KUKA KRL program: MyProgram_016().src

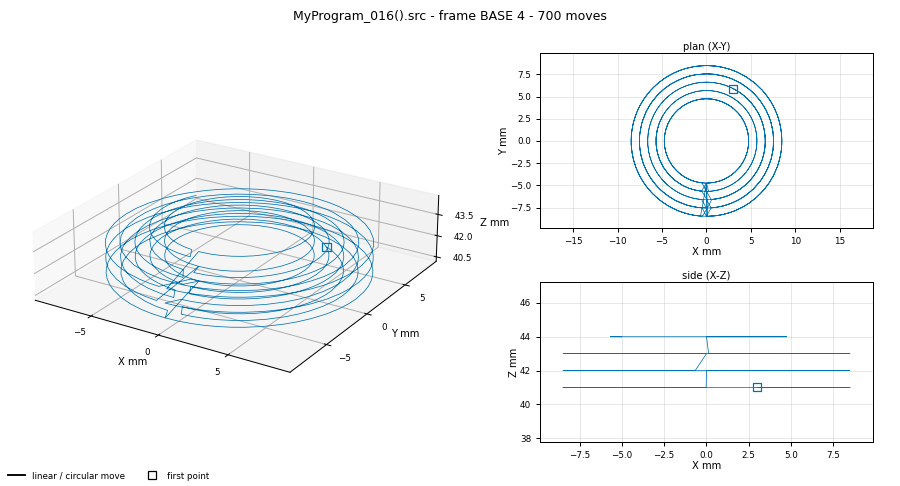
[picture p0: tool path of MyProgram_016().src in frame BASE 4, 700 of 700 moves have a stored position in this frame; points joined in program order, loops and branches not executed]
&ACCESS RVP
&REL 1
&PARAM TEMPLATE = C:\KRC\Roboter\Template\vorgabe
&PARAM EDITMASK = *
DEF MyProgram_016()
; ---- Setting reference (Base) ----
$BASE = BASE_DATA[4]

; --------------------------
; ---- Setting tool (TCP) ----
$TOOL = TOOL_DATA[3]
; --------------------------

$VEL.CP = VEL_APROX_PRINT
Startdeposition()
$VEL.CP = VEL_PRINT
LIN {X 3.0027,Y 5.8982,Z 41,A -2.319,B 0,C 0,E1 0.1598,E2 90.0724} C_DIS
LIN {X 3.6295,Y 5.5354,Z 41,A -2.3113,B 0,C 0,E1 0.1598,E2 90.0724} C_DIS
LIN {X 4.2131,Y 5.1066,Z 41,A -2.308,B 0,C 0,E1 0.1598,E2 90.0724} C_DIS
LIN {X 4.7456,Y 4.6156,Z 41,A -2.3092,B 0,C 0,E1 0.1598,E2 90.0724} C_DIS
LIN {X 5.2207,Y 4.0691,Z 41,A -2.3149,B 0,C 0,E1 0.1598,E2 90.0723} C_DIS
LIN {X 5.6347,Y 3.4746,Z 41,A -2.3249,B 0,C 0,E1 0.1598,E2 90.0723} C_DIS
LIN {X 5.9818,Y 2.8391,Z 41,A -2.3392,B 0,C 0,E1 0.1598,E2 90.0723} C_DIS
LIN {X 6.2545,Y 2.1682,Z 41,A -2.3577,B 0,C 0,E1 0.1598,E2 90.0722} C_DIS
LIN {X 6.4955,Y 1.2955,Z 41,A -2.3857,B 0,C 0,E1 0.1598,E2 90.0719} C_DIS
LIN {X 6.6144,Y 0.2312,Z 41,A -2.4266,B 0,C 0,E1 0.1598,E2 90.0717} C_DIS
LIN {X 6.5984,Y -0.514,Z 41,A -2.4593,B 0,C 0,E1 0.1598,E2 90.072} C_DIS
LIN {X 6.4986,Y -1.2526,Z 41,A -2.4944,B 0,C 0,E1 0.1598,E2 90.072} C_DIS
LIN {X 6.3195,Y -1.9763,Z 41,A -2.5319,B 0,C 0,E1 0.1598,E2 90.072} C_DIS
LIN {X 6.0549,Y -2.6732,Z 41,A -2.5714,B 0,C 0,E1 0.1598,E2 90.0719} C_DIS
LIN {X 5.7165,Y -3.3374,Z 41,A -2.6122,B 0,C 0,E1 0.1598,E2 90.0719} C_DIS
LIN {X 5.3054,Y -3.9593,Z 41,A -2.6538,B 0,C 0,E1 0.1598,E2 90.0719} C_DIS
LIN {X 4.8275,Y -4.5316,Z 41,A -2.6958,B 0,C 0,E1 0.1598,E2 90.0719} C_DIS
LIN {X 4.2857,Y -5.0436,Z 41,A -2.7375,B 0,C 0,E1 0.1598,E2 90.0718} C_DIS
LIN {X 3.691,Y -5.4931,Z 41,A -2.7785,B 0,C 0,E1 0.1598,E2 90.0718} C_DIS
LIN {X 3.0503,Y -5.874,Z 41,A -2.8183,B 0,C 0,E1 0.1598,E2 90.0718} C_DIS
LIN {X 2.3699,Y -6.1782,Z 41,A -2.8563,B 0,C 0,E1 0.1598,E2 90.0718} C_DIS
LIN {X 1.6605,Y -6.4069,Z 41,A -2.892,B 0,C 0,E1 0.1598,E2 90.0717} C_DIS
LIN {X 0.9297,Y -6.5533,Z 41,A -2.9251,B 0,C 0,E1 0.1598,E2 90.0717} C_DIS
LIN {X 0.0006,Y -6.6224,Z 41,A -2.9621,B 0,C 0,E1 0.1598,E2 90.0717} C_DIS
Enddeposition()
LIN {X 0.0006,Y -6.6224,Z 41,A -2.9621,B 0,C 0,E1 0.1598,E2 90.0717} C_DIS
Startdeposition()
$VEL.CP = VEL_PRINT
LIN {X 0.5218,Y -7.5346,Z 41,A -2.9814,B 0,C 0,E1 0.1598,E2 90.071} C_DIS
LIN {X 1.2142,Y -7.4561,Z 41,A -2.9532,B 0,C 0,E1 0.1598,E2 90.0716} C_DIS
LIN {X 1.8961,Y -7.3127,Z 41,A -2.9222,B 0,C 0,E1 0.1598,E2 90.0716} C_DIS
LIN {X 2.7263,Y -7.0488,Z 41,A -2.8805,B 0,C 0,E1 0.1598,E2 90.0716} C_DIS
LIN {X 3.6839,Y -6.5978,Z 41,A -2.8261,B 0,C 0,E1 0.1598,E2 90.0717} C_DIS
LIN {X 4.3969,Y -6.1467,Z 41,A -2.7807,B 0,C 0,E1 0.1598,E2 90.0717} C_DIS
LIN {X 5.2728,Y -5.4135,Z 41,A -2.7171,B 0,C 0,E1 0.1598,E2 90.0717} C_DIS
LIN {X 6.0845,Y -4.4837,Z 41,A -2.6475,B 0,C 0,E1 0.1598,E2 90.0717} C_DIS
LIN {X 6.5832,Y -3.7041,Z 41,A -2.596,B 0,C 0,E1 0.1598,E2 90.0718} C_DIS
LIN {X 6.9129,Y -3.0412,Z 41,A -2.5557,B 0,C 0,E1 0.1598,E2 90.0719} C_DIS
LIN {X 7.287,Y -2.0035,Z 41,A -2.4973,B 0,C 0,E1 0.1598,E2 90.0717} C_DIS
LIN {X 7.4913,Y -1.0048,Z 41,A -2.4471,B 0,C 0,E1 0.1598,E2 90.0717} C_DIS
LIN {X 7.5586,Y -0.0079,Z 41,A -2.4022,B 0,C 0,E1 0.1598,E2 90.0718} C_DIS
LIN {X 7.499,Y 0.937,Z 41,A -2.3641,B 0,C 0,E1 0.1598,E2 90.0719} C_DIS
LIN {X 7.2647,Y 2.068,Z 41,A -2.3242,B 0,C 0,E1 0.1598,E2 90.0717} C_DIS
LIN {X 7.0052,Y 2.8257,Z 41,A -2.3019,B 0,C 0,E1 0.1598,E2 90.0721} C_DIS
LIN {X 6.6657,Y 3.5511,Z 41,A -2.2835,B 0,C 0,E1 0.1598,E2 90.0722} C_DIS
LIN {X 6.0442,Y 4.5361,Z 41,A -2.2642,B 0,C 0,E1 0.1598,E2 90.072} C_DIS
LIN {X 5.3435,Y 5.346,Z 41,A -2.2557,B 0,C 0,E1 0.1598,E2 90.0722} C_DIS
LIN {X 4.6544,Y 5.9486,Z 41,A -2.2557,B 0,C 0,E1 0.1598,E2 90.0723} C_DIS
LIN {X 3.7373,Y 6.5685,Z 41,A -2.2631,B 0,C 0,E1 0.1598,E2 90.0723} C_DIS
LIN {X 2.7804,Y 7.0216,Z 41,A -2.2793,B 0,C 0,E1 0.1598,E2 90.0723} C_DIS
LIN {X 1.9771,Y 7.2898,Z 41,A -2.2976,B 0,C 0,E1 0.1598,E2 90.0725} C_DIS
LIN {X 0.8628,Y 7.5074,Z 41,A -2.3295,B 0,C 0,E1 0.1598,E2 90.0725} C_DIS
LIN {X -0.0807,Y 7.557,Z 41,A -2.3623,B 0,C 0,E1 0.1598,E2 90.0725} C_DIS
LIN {X -1.2554,Y 7.4477,Z 41,A -2.4103,B 0,C 0,E1 0.1598,E2 90.0724} C_DIS
LIN {X -2.007,Y 7.2809,Z 41,A -2.4451,B 0,C 0,E1 0.1598,E2 90.0723} C_DIS
LIN {X -2.7375,Y 7.0382,Z 41,A -2.4823,B 0,C 0,E1 0.1598,E2 90.0723} C_DIS
LIN {X -3.9575,Y 6.4373,Z 41,A -2.5526,B 0,C 0,E1 0.1598,E2 90.072} C_DIS
LIN {X -4.6822,Y 5.9317,Z 41,A -2.6008,B 0,C 0,E1 0.1598,E2 90.072} C_DIS
LIN {X -5.4823,Y 5.2003,Z 41,A -2.6611,B 0,C 0,E1 0.1598,E2 90.0718} C_DIS
LIN {X -6.1884,Y 4.3366,Z 41,A -2.7235,B 0,C 0,E1 0.1598,E2 90.0716} C_DIS
LIN {X -6.7771,Y 3.3427,Z 41,A -2.7871,B 0,C 0,E1 0.1598,E2 90.0714} C_DIS
LIN {X -7.2905,Y 1.9898,Z 41,A -2.8628,B 0,C 0,E1 0.1598,E2 90.0708} C_DIS
LIN {X -7.5205,Y 0.6986,Z 41,A -2.9259,B 0,C 0,E1 0.1598,E2 90.0708} C_DIS
LIN {X -7.5526,Y -0.1182,Z 41,A -2.9621,B 0,C 0,E1 0.1598,E2 90.0712} C_DIS
LIN {X -7.4933,Y -0.9334,Z 41,A -2.9944,B 0,C 0,E1 0.1598,E2 90.0712} C_DIS
LIN {X -7.3508,Y -1.7381,Z 41,A -3.0233,B 0,C 0,E1 0.1598,E2 90.0712} C_DIS
LIN {X -7.0039,Y -2.8395,Z 41,A -3.0569,B 0,C 0,E1 0.1598,E2 90.0709} C_DIS
LIN {X -6.6343,Y -3.6177,Z 41,A -3.0765,B 0,C 0,E1 0.1598,E2 90.0712} C_DIS
LIN {X -5.9525,Y -4.6552,Z 41,A -3.0952,B 0,C 0,E1 0.1598,E2 90.0708} C_DIS
LIN {X -5.2119,Y -5.4671,Z 41,A -3.1027,B 0,C 0,E1 0.1598,E2 90.0711} C_DIS
LIN {X -4.6479,Y -5.9517,Z 41,A -3.1027,B 0,C 0,E1 0.1598,E2 90.0713} C_DIS
LIN {X -4.0412,Y -6.3817,Z 41,A -3.0988,B 0,C 0,E1 0.1598,E2 90.0713} C_DIS
LIN {X -3.394,Y -6.7479,Z 41,A -3.0906,B 0,C 0,E1 0.1598,E2 90.0713} C_DIS
LIN {X -2.388,Y -7.1707,Z 41,A -3.0717,B 0,C 0,E1 0.1598,E2 90.0713} C_DIS
LIN {X -1.4895,Y -7.4088,Z 41,A -3.0489,B 0,C 0,E1 0.1598,E2 90.0715} C_DIS
LIN {X -0.4781,Y -7.5384,Z 41,A -3.0174,B 0,C 0,E1 0.1598,E2 90.0715} C_DIS
LIN {X -0.4781,Y -7.5384,Z 41,A -3.0174,B 0,C 0,E1 0.1598,E2 90.0715} C_DIS
Enddeposition()
LIN {X -0.0182,Y -8.489,Z 41,A -3.04,B 0,C 0,E1 0.1598,E2 90.0703} C_DIS
Startdeposition()
$VEL.CP = VEL_PRINT
LIN {X -1.0751,Y -8.4193,Z 41,A -3.0769,B 0,C 0,E1 0.1598,E2 90.0714} C_DIS
LIN {X -1.9094,Y -8.27,Z 41,A -3.1012,B 0,C 0,E1 0.1598,E2 90.0714} C_DIS
LIN {X -2.9255,Y -7.9703,Z 41,A -3.1256,B 0,C 0,E1 0.1598,E2 90.0714} C_DIS
LIN {X -3.9562,Y -7.5135,Z 41,A -3.1439,B 0,C 0,E1 0.1598,E2 90.0712} C_DIS
LIN {X -5.0038,Y -6.8555,Z 41,A -3.1543,B 0,C 0,E1 0.1598,E2 90.0712} C_DIS
LIN {X -5.667,Y -6.3182,Z 41,A -3.1559,B 0,C 0,E1 0.1598,E2 90.0712} C_DIS
LIN {X -6.273,Y -5.7172,Z 41,A -3.1526,B 0,C 0,E1 0.1598,E2 90.0712} C_DIS
LIN {X -6.8156,Y -5.0583,Z 41,A -3.1445,B 0,C 0,E1 0.1598,E2 90.0712} C_DIS
LIN {X -7.2893,Y -4.3483,Z 41,A -3.1318,B 0,C 0,E1 0.1598,E2 90.0712} C_DIS
LIN {X -7.6893,Y -3.5943,Z 41,A -3.1145,B 0,C 0,E1 0.1598,E2 90.0712} C_DIS
LIN {X -8.0114,Y -2.8039,Z 41,A -3.0929,B 0,C 0,E1 0.1598,E2 90.0712} C_DIS
LIN {X -8.2523,Y -1.9851,Z 41,A -3.0671,B 0,C 0,E1 0.1598,E2 90.0712} C_DIS
LIN {X -8.4389,Y -0.9347,Z 41,A -3.0292,B 0,C 0,E1 0.1598,E2 90.0709} C_DIS
LIN {X -8.4896,Y 0.137,Z 41,A -2.9857,B 0,C 0,E1 0.1598,E2 90.0709} C_DIS
LIN {X -8.4116,Y 1.1667,Z 41,A -2.9394,B 0,C 0,E1 0.1598,E2 90.0711} C_DIS
LIN {X -8.1845,Y 2.2482,Z 41,A -2.8853,B 0,C 0,E1 0.1598,E2 90.0711} C_DIS
LIN {X -7.7971,Y 3.36,Z 41,A -2.824,B 0,C 0,E1 0.1598,E2 90.0712} C_DIS
LIN {X -7.21,Y 4.483,Z 41,A -2.7549,B 0,C 0,E1 0.1598,E2 90.0712} C_DIS
LIN {X -6.5678,Y 5.3748,Z 41,A -2.6937,B 0,C 0,E1 0.1598,E2 90.0716} C_DIS
LIN {X -5.9685,Y 6.0403,Z 41,A -2.6436,B 0,C 0,E1 0.1598,E2 90.0718} C_DIS
LIN {X -5.0746,Y 6.8036,Z 41,A -2.5784,B 0,C 0,E1 0.1598,E2 90.0718} C_DIS
LIN {X -4.3639,Y 7.2802,Z 41,A -2.5321,B 0,C 0,E1 0.1598,E2 90.0721} C_DIS
LIN {X -3.6087,Y 7.6827,Z 41,A -2.4873,B 0,C 0,E1 0.1598,E2 90.0721} C_DIS
LIN {X -2.8167,Y 8.0069,Z 41,A -2.4444,B 0,C 0,E1 0.1598,E2 90.0723} C_DIS
LIN {X -1.9961,Y 8.2497,Z 41,A -2.4038,B 0,C 0,E1 0.1598,E2 90.0723} C_DIS
LIN {X -1.1553,Y 8.4087,Z 41,A -2.366,B 0,C 0,E1 0.1598,E2 90.0724} C_DIS
LIN {X -0.0888,Y 8.4907,Z 41,A -2.3232,B 0,C 0,E1 0.1598,E2 90.0724} C_DIS
LIN {X 1.0545,Y 8.4223,Z 41,A -2.2839,B 0,C 0,E1 0.1598,E2 90.0725} C_DIS
LIN {X 1.8987,Y 8.2723,Z 41,A -2.2591,B 0,C 0,E1 0.1598,E2 90.0725} C_DIS
LIN {X 2.7237,Y 8.0385,Z 41,A -2.2385,B 0,C 0,E1 0.1598,E2 90.0725} C_DIS
LIN {X 3.5208,Y 7.7226,Z 41,A -2.2225,B 0,C 0,E1 0.1598,E2 90.0725} C_DIS
LIN {X 4.4673,Y 7.2197,Z 41,A -2.2088,B 0,C 0,E1 0.1598,E2 90.0725} C_DIS
LIN {X 5.5023,Y 6.4657,Z 41,A -2.2025,B 0,C 0,E1 0.1598,E2 90.0723} C_DIS
LIN {X 6.2699,Y 5.7205,Z 41,A -2.2059,B 0,C 0,E1 0.1598,E2 90.0723} C_DIS
LIN {X 6.8143,Y 5.0601,Z 41,A -2.214,B 0,C 0,E1 0.1598,E2 90.0723} C_DIS
LIN {X 7.2893,Y 4.3481,Z 41,A -2.2268,B 0,C 0,E1 0.1598,E2 90.0723} C_DIS
LIN {X 7.6903,Y 3.592,Z 41,A -2.2442,B 0,C 0,E1 0.1598,E2 90.0723} C_DIS
LIN {X 8.0125,Y 2.7991,Z 41,A -2.2661,B 0,C 0,E1 0.1598,E2 90.0722} C_DIS
LIN {X 8.2538,Y 1.978,Z 41,A -2.2922,B 0,C 0,E1 0.1598,E2 90.0722} C_DIS
LIN {X 8.4112,Y 1.1367,Z 41,A -2.3223,B 0,C 0,E1 0.1598,E2 90.0721} C_DIS
LIN {X 8.4922,Y -0.0058,Z 41,A -2.3678,B 0,C 0,E1 0.1598,E2 90.0717} C_DIS
LIN {X 8.4473,Y -0.8607,Z 41,A -2.406,B 0,C 0,E1 0.1598,E2 90.0717} C_DIS
LIN {X 8.3172,Y -1.7063,Z 41,A -2.4471,B 0,C 0,E1 0.1598,E2 90.0719} C_DIS
LIN {X 8.0233,Y -2.7811,Z 41,A -2.5036,B 0,C 0,E1 0.1598,E2 90.0717} C_DIS
LIN {X 7.5387,Y -3.8974,Z 41,A -2.5689,B 0,C 0,E1 0.1598,E2 90.0714} C_DIS
LIN {X 7.0759,Y -4.6845,Z 41,A -2.6199,B 0,C 0,E1 0.1598,E2 90.0717} C_DIS
LIN {X 6.5318,Y -5.4179,Z 41,A -2.6712,B 0,C 0,E1 0.1598,E2 90.0717} C_DIS
LIN {X 5.6483,Y -6.3408,Z 41,A -2.7429,B 0,C 0,E1 0.1598,E2 90.0715} C_DIS
LIN {X 4.7399,Y -7.0403,Z 41,A -2.8062,B 0,C 0,E1 0.1598,E2 90.0715} C_DIS
LIN {X 4.0492,Y -7.4582,Z 41,A -2.8495,B 0,C 0,E1 0.1598,E2 90.0717} C_DIS
LIN {X 3.3221,Y -7.8087,Z 41,A -2.8911,B 0,C 0,E1 0.1598,E2 90.0717} C_DIS
LIN {X 2.5651,Y -8.0886,Z 41,A -2.9308,B 0,C 0,E1 0.1598,E2 90.0717} C_DIS
LIN {X 1.785,Y -8.2955,Z 41,A -2.9683,B 0,C 0,E1 0.1598,E2 90.0717} C_DIS
LIN {X 0.9888,Y -8.4278,Z 41,A -3.0031,B 0,C 0,E1 0.1598,E2 90.0716} C_DIS
LIN {X -0.0182,Y -8.489,Z 41,A -3.0426,B 0,C 0,E1 0.1598,E2 90.0716} C_DIS
Enddeposition()
LIN {X 0.0009,Y -4.7546,Z 42,A -2.8683,B 0,C 0,E1 0.1598,E2 90.0604} C_DIS
Startdeposition()
$VEL.CP = VEL_PRINT
LIN {X 0.0009,Y -4.7546,Z 42,A -2.8741,B 0,C 0,E1 0.1598,E2 90.0661} C_DIS
LIN {X 0.8353,Y -4.6792,Z 42,A -2.8451,B 0,C 0,E1 0.1598,E2 90.0711} C_DIS
LIN {X 1.4852,Y -4.5142,Z 42,A -2.8149,B 0,C 0,E1 0.1598,E2 90.0718} C_DIS
LIN {X 2.1053,Y -4.2593,Z 42,A -2.7813,B 0,C 0,E1 0.1598,E2 90.0718} C_DIS
LIN {X 2.7516,Y -3.8714,Z 42,A -2.741,B 0,C 0,E1 0.1598,E2 90.0718} C_DIS
LIN {X 3.2075,Y -3.5024,Z 42,A -2.7085,B 0,C 0,E1 0.1598,E2 90.0719} C_DIS
LIN {X 3.671,Y -3.0181,Z 42,A -2.6708,B 0,C 0,E1 0.1598,E2 90.0719} C_DIS
LIN {X 4.0596,Y -2.4718,Z 42,A -2.6332,B 0,C 0,E1 0.1598,E2 90.0719} C_DIS
LIN {X 4.3647,Y -1.8749,Z 42,A -2.5966,B 0,C 0,E1 0.1598,E2 90.0719} C_DIS
LIN {X 4.5854,Y -1.2421,Z 42,A -2.5614,B 0,C 0,E1 0.1598,E2 90.0719} C_DIS
LIN {X 4.7151,Y -0.5846,Z 42,A -2.5286,B 0,C 0,E1 0.1598,E2 90.0719} C_DIS
LIN {X 4.7506,Y 0.0847,Z 42,A -2.4988,B 0,C 0,E1 0.1598,E2 90.0719} C_DIS
LIN {X 4.6913,Y 0.7523,Z 42,A -2.4725,B 0,C 0,E1 0.1598,E2 90.072} C_DIS
LIN {X 4.539,Y 1.405,Z 42,A -2.4504,B 0,C 0,E1 0.1598,E2 90.072} C_DIS
LIN {X 4.2971,Y 2.0303,Z 42,A -2.4327,B 0,C 0,E1 0.1598,E2 90.072} C_DIS
LIN {X 3.9682,Y 2.6145,Z 42,A -2.4199,B 0,C 0,E1 0.1598,E2 90.0721} C_DIS
LIN {X 3.5592,Y 3.1456,Z 42,A -2.4124,B 0,C 0,E1 0.1598,E2 90.0721} C_DIS
LIN {X 3.0809,Y 3.6151,Z 42,A -2.4101,B 0,C 0,E1 0.1598,E2 90.0722} C_DIS
LIN {X 2.5429,Y 4.0149,Z 42,A -2.413,B 0,C 0,E1 0.1598,E2 90.0722} C_DIS
LIN {X 1.8748,Y 4.3642,Z 42,A -2.4228,B 0,C 0,E1 0.1598,E2 90.0722} C_DIS
LIN {X 1.3227,Y 4.562,Z 42,A -2.4348,B 0,C 0,E1 0.1598,E2 90.0722} C_DIS
LIN {X 0.6678,Y 4.7047,Z 42,A -2.4529,B 0,C 0,E1 0.1598,E2 90.0722} C_DIS
LIN {X -0.0009,Y 4.7506,Z 42,A -2.4756,B 0,C 0,E1 0.1598,E2 90.0722} C_DIS
LIN {X -0.6694,Y 4.7033,Z 42,A -2.5022,B 0,C 0,E1 0.1598,E2 90.0722} C_DIS
LIN {X -1.3245,Y 4.5621,Z 42,A -2.5324,B 0,C 0,E1 0.1598,E2 90.0722} C_DIS
LIN {X -1.9536,Y 4.331,Z 42,A -2.5653,B 0,C 0,E1 0.1598,E2 90.0722} C_DIS
LIN {X -2.5432,Y 4.0123,Z 42,A -2.6005,B 0,C 0,E1 0.1598,E2 90.0721} C_DIS
LIN {X -3.0824,Y 3.6143,Z 42,A -2.6372,B 0,C 0,E1 0.1598,E2 90.072} C_DIS
LIN {X -3.561,Y 3.145,Z 42,A -2.6747,B 0,C 0,E1 0.1598,E2 90.0719} C_DIS
LIN {X -3.9685,Y 2.6128,Z 42,A -2.7122,B 0,C 0,E1 0.1598,E2 90.0719} C_DIS
LIN {X -4.2978,Y 2.0289,Z 42,A -2.7491,B 0,C 0,E1 0.1598,E2 90.0717} C_DIS
LIN {X -4.5408,Y 1.404,Z 42,A -2.7845,B 0,C 0,E1 0.1598,E2 90.0717} C_DIS
LIN {X -4.6932,Y 0.7511,Z 42,A -2.8177,B 0,C 0,E1 0.1598,E2 90.0716} C_DIS
LIN {X -4.7509,Y 0.0831,Z 42,A -2.8481,B 0,C 0,E1 0.1598,E2 90.0716} C_DIS
LIN {X -4.7165,Y -0.5864,Z 42,A -2.8752,B 0,C 0,E1 0.1598,E2 90.0716} C_DIS
LIN {X -4.5857,Y -1.2439,Z 42,A -2.8983,B 0,C 0,E1 0.1598,E2 90.0715} C_DIS
LIN {X -4.3651,Y -1.8769,Z 42,A -2.917,B 0,C 0,E1 0.1598,E2 90.0715} C_DIS
LIN {X -4.056,Y -2.4715,Z 42,A -2.9309,B 0,C 0,E1 0.1598,E2 90.0715} C_DIS
LIN {X -3.6697,Y -3.0195,Z 42,A -2.94,B 0,C 0,E1 0.1598,E2 90.0715} C_DIS
LIN {X -3.2069,Y -3.5044,Z 42,A -2.9436,B 0,C 0,E1 0.1598,E2 90.0715} C_DIS
LIN {X -2.6822,Y -3.9215,Z 42,A -2.9421,B 0,C 0,E1 0.1598,E2 90.0715} C_DIS
LIN {X -2.103,Y -4.2589,Z 42,A -2.9352,B 0,C 0,E1 0.1598,E2 90.0715} C_DIS
LIN {X -1.4832,Y -4.5137,Z 42,A -2.9233,B 0,C 0,E1 0.1598,E2 90.0716} C_DIS
LIN {X -0.8333,Y -4.6776,Z 42,A -2.9064,B 0,C 0,E1 0.1598,E2 90.0716} C_DIS
LIN {X 0.0009,Y -4.7546,Z 42,A -2.8791,B 0,C 0,E1 0.1598,E2 90.0717} C_DIS
Enddeposition()
LIN {X 0.0009,Y -4.7546,Z 42,A -2.8791,B 0,C 0,E1 0.1598,E2 90.0717} C_DIS
Startdeposition()
$VEL.CP = VEL_PRINT
LIN {X -0.5645,Y -5.6544,Z 42,A -2.9376,B 0,C 0,E1 0.1598,E2 90.0711} C_DIS
LIN {X -1.3254,Y -5.5269,Z 42,A -2.9607,B 0,C 0,E1 0.1598,E2 90.0716} C_DIS
LIN {X -2.0618,Y -5.2961,Z 42,A -2.9779,B 0,C 0,E1 0.1598,E2 90.0716} C_DIS
LIN {X -2.7614,Y -4.9704,Z 42,A -2.9897,B 0,C 0,E1 0.1598,E2 90.0716} C_DIS
LIN {X -3.7147,Y -4.3091,Z 42,A -2.9964,B 0,C 0,E1 0.1598,E2 90.0713} C_DIS
LIN {X -4.194,Y -3.8378,Z 42,A -2.9941,B 0,C 0,E1 0.1598,E2 90.0714} C_DIS
LIN {X -4.748,Y -3.1366,Z 42,A -2.9844,B 0,C 0,E1 0.1598,E2 90.0712} C_DIS
LIN {X -5.0695,Y -2.571,Z 42,A -2.9725,B 0,C 0,E1 0.1598,E2 90.0714} C_DIS
LIN {X -5.4016,Y -1.7705,Z 42,A -2.9506,B 0,C 0,E1 0.1598,E2 90.0713} C_DIS
LIN {X -5.6083,Y -0.9288,Z 42,A -2.9225,B 0,C 0,E1 0.1598,E2 90.0713} C_DIS
LIN {X -5.6835,Y -0.2826,Z 42,A -2.8981,B 0,C 0,E1 0.1598,E2 90.0715} C_DIS
LIN {X -5.6648,Y 0.4908,Z 42,A -2.8646,B 0,C 0,E1 0.1598,E2 90.0715} C_DIS
LIN {X -5.5348,Y 1.2885,Z 42,A -2.8259,B 0,C 0,E1 0.1598,E2 90.0715} C_DIS
LIN {X -5.2959,Y 2.0604,Z 42,A -2.7845,B 0,C 0,E1 0.1598,E2 90.0715} C_DIS
LIN {X -4.9503,Y 2.7907,Z 42,A -2.7409,B 0,C 0,E1 0.1598,E2 90.0716} C_DIS
LIN {X -4.5058,Y 3.4656,Z 42,A -2.696,B 0,C 0,E1 0.1598,E2 90.0717} C_DIS
LIN {X -3.9695,Y 4.0704,Z 42,A -2.6506,B 0,C 0,E1 0.1598,E2 90.0719} C_DIS
LIN {X -3.3518,Y 4.5918,Z 42,A -2.6058,B 0,C 0,E1 0.1598,E2 90.0719} C_DIS
LIN {X -2.396,Y 5.1611,Z 42,A -2.5465,B 0,C 0,E1 0.1598,E2 90.072} C_DIS
LIN {X -1.1034,Y 5.5819,Z 42,A -2.481,B 0,C 0,E1 0.1598,E2 90.0722} C_DIS
LIN {X -0.0792,Y 5.684,Z 42,A -2.439,B 0,C 0,E1 0.1598,E2 90.0723} C_DIS
LIN {X 0.7426,Y 5.6348,Z 42,A -2.4108,B 0,C 0,E1 0.1598,E2 90.0723} C_DIS
LIN {X 1.5485,Y 5.4674,Z 42,A -2.3882,B 0,C 0,E1 0.1598,E2 90.0723} C_DIS
LIN {X 2.322,Y 5.1863,Z 42,A -2.3715,B 0,C 0,E1 0.1598,E2 90.0723} C_DIS
LIN {X 3.0471,Y 4.7968,Z 42,A -2.3613,B 0,C 0,E1 0.1598,E2 90.0723} C_DIS
LIN {X 3.7088,Y 4.307,Z 42,A -2.3577,B 0,C 0,E1 0.1598,E2 90.0723} C_DIS
LIN {X 4.2923,Y 3.7262,Z 42,A -2.3609,B 0,C 0,E1 0.1598,E2 90.0723} C_DIS
LIN {X 4.7867,Y 3.0677,Z 42,A -2.3706,B 0,C 0,E1 0.1598,E2 90.0721} C_DIS
LIN {X 5.1788,Y 2.3435,Z 42,A -2.387,B 0,C 0,E1 0.1598,E2 90.0721} C_DIS
LIN {X 5.462,Y 1.5704,Z 42,A -2.4094,B 0,C 0,E1 0.1598,E2 90.0721} C_DIS
LIN {X 5.6334,Y 0.7652,Z 42,A -2.4374,B 0,C 0,E1 0.1598,E2 90.0719} C_DIS
LIN {X 5.6827,Y -0.0566,Z 42,A -2.4706,B 0,C 0,E1 0.1598,E2 90.0719} C_DIS
LIN {X 5.6151,Y -0.877,Z 42,A -2.508,B 0,C 0,E1 0.1598,E2 90.0719} C_DIS
LIN {X 5.4319,Y -1.6797,Z 42,A -2.549,B 0,C 0,E1 0.1598,E2 90.0719} C_DIS
LIN {X 5.1314,Y -2.4463,Z 42,A -2.5928,B 0,C 0,E1 0.1598,E2 90.0718} C_DIS
LIN {X 4.7229,Y -3.1611,Z 42,A -2.6383,B 0,C 0,E1 0.1598,E2 90.0718} C_DIS
LIN {X 4.2175,Y -3.811,Z 42,A -2.6846,B 0,C 0,E1 0.1598,E2 90.0718} C_DIS
LIN {X 3.6236,Y -4.3814,Z 42,A -2.7308,B 0,C 0,E1 0.1598,E2 90.0718} C_DIS
LIN {X 2.9526,Y -4.8589,Z 42,A -2.7758,B 0,C 0,E1 0.1598,E2 90.0718} C_DIS
LIN {X 2.2189,Y -5.2329,Z 42,A -2.8187,B 0,C 0,E1 0.1598,E2 90.0718} C_DIS
LIN {X 1.4397,Y -5.4984,Z 42,A -2.8586,B 0,C 0,E1 0.1598,E2 90.0718} C_DIS
LIN {X 0.6301,Y -5.6475,Z 42,A -2.8947,B 0,C 0,E1 0.1598,E2 90.0718} C_DIS
LIN {X 0.0136,Y -5.6876,Z 42,A -2.919,B 0,C 0,E1 0.1598,E2 90.0717} C_DIS
Enddeposition()
LIN {X 0.0136,Y -5.6876,Z 42,A -2.919,B 0,C 0,E1 0.1598,E2 90.0717} C_DIS
Startdeposition()
$VEL.CP = VEL_PRINT
LIN {X 0.5245,Y -6.6006,Z 42,A -2.9387,B 0,C 0,E1 0.1598,E2 90.0711} C_DIS
LIN {X 1.2172,Y -6.5067,Z 42,A -2.9099,B 0,C 0,E1 0.1598,E2 90.0717} C_DIS
LIN {X 1.8962,Y -6.3409,Z 42,A -2.8779,B 0,C 0,E1 0.1598,E2 90.0717} C_DIS
LIN {X 2.5549,Y -6.1067,Z 42,A -2.8438,B 0,C 0,E1 0.1598,E2 90.0717} C_DIS
LIN {X 3.1844,Y -5.8028,Z 42,A -2.8077,B 0,C 0,E1 0.1598,E2 90.0717} C_DIS
LIN {X 3.7779,Y -5.4336,Z 42,A -2.7702,B 0,C 0,E1 0.1598,E2 90.0718} C_DIS
LIN {X 4.3301,Y -5.0052,Z 42,A -2.7316,B 0,C 0,E1 0.1598,E2 90.0718} C_DIS
LIN {X 4.8359,Y -4.5227,Z 42,A -2.6924,B 0,C 0,E1 0.1598,E2 90.0718} C_DIS
LIN {X 5.2851,Y -3.9869,Z 42,A -2.6531,B 0,C 0,E1 0.1598,E2 90.0718} C_DIS
LIN {X 5.6761,Y -3.4074,Z 42,A -2.614,B 0,C 0,E1 0.1598,E2 90.0719} C_DIS
LIN {X 6.0039,Y -2.7899,Z 42,A -2.5756,B 0,C 0,E1 0.1598,E2 90.0719} C_DIS
LIN {X 6.2645,Y -2.1412,Z 42,A -2.5383,B 0,C 0,E1 0.1598,E2 90.0719} C_DIS
LIN {X 6.4557,Y -1.4689,Z 42,A -2.5025,B 0,C 0,E1 0.1598,E2 90.0719} C_DIS
LIN {X 6.5739,Y -0.7799,Z 42,A -2.4688,B 0,C 0,E1 0.1598,E2 90.072} C_DIS
LIN {X 6.6171,Y -0.0824,Z 42,A -2.4374,B 0,C 0,E1 0.1598,E2 90.072} C_DIS
LIN {X 6.576,Y 0.7905,Z 42,A -2.4015,B 0,C 0,E1 0.1598,E2 90.0719} C_DIS
LIN {X 6.3641,Y 1.8191,Z 42,A -2.3653,B 0,C 0,E1 0.1598,E2 90.0718} C_DIS
LIN {X 6.1307,Y 2.5001,Z 42,A -2.3452,B 0,C 0,E1 0.1598,E2 90.0721} C_DIS
LIN {X 5.8236,Y 3.1513,Z 42,A -2.3288,B 0,C 0,E1 0.1598,E2 90.0722} C_DIS
LIN {X 5.4439,Y 3.7629,Z 42,A -2.3168,B 0,C 0,E1 0.1598,E2 90.0722} C_DIS
LIN {X 5.0047,Y 4.3334,Z 42,A -2.3087,B 0,C 0,E1 0.1598,E2 90.0722} C_DIS
LIN {X 4.5044,Y 4.851,Z 42,A -2.3052,B 0,C 0,E1 0.1598,E2 90.0723} C_DIS
LIN {X 3.951,Y 5.3115,Z 42,A -2.306,B 0,C 0,E1 0.1598,E2 90.0723} C_DIS
LIN {X 3.3506,Y 5.7087,Z 42,A -2.3113,B 0,C 0,E1 0.1598,E2 90.0723} C_DIS
LIN {X 2.7108,Y 6.0389,Z 42,A -2.3209,B 0,C 0,E1 0.1598,E2 90.0724} C_DIS
LIN {X 2.0384,Y 6.2962,Z 42,A -2.3348,B 0,C 0,E1 0.1598,E2 90.0724} C_DIS
LIN {X 1.343,Y 6.4824,Z 42,A -2.3526,B 0,C 0,E1 0.1598,E2 90.0724} C_DIS
LIN {X 0.6308,Y 6.5873,Z 42,A -2.3744,B 0,C 0,E1 0.1598,E2 90.0724} C_DIS
LIN {X -0.0885,Y 6.6195,Z 42,A -2.3996,B 0,C 0,E1 0.1598,E2 90.0724} C_DIS
LIN {X -0.8068,Y 6.5719,Z 42,A -2.4281,B 0,C 0,E1 0.1598,E2 90.0724} C_DIS
LIN {X -1.5154,Y 6.4439,Z 42,A -2.4597,B 0,C 0,E1 0.1598,E2 90.0723} C_DIS
LIN {X -2.206,Y 6.2406,Z 42,A -2.4937,B 0,C 0,E1 0.1598,E2 90.0723} C_DIS
LIN {X -2.8706,Y 5.9638,Z 42,A -2.53,B 0,C 0,E1 0.1598,E2 90.0722} C_DIS
LIN {X -3.5019,Y 5.6178,Z 42,A -2.5679,B 0,C 0,E1 0.1598,E2 90.0721} C_DIS
LIN {X -4.0918,Y 5.2049,Z 42,A -2.6071,B 0,C 0,E1 0.1598,E2 90.0721} C_DIS
LIN {X -4.6325,Y 4.7294,Z 42,A -2.6471,B 0,C 0,E1 0.1598,E2 90.0719} C_DIS
LIN {X -5.118,Y 4.1976,Z 42,A -2.6875,B 0,C 0,E1 0.1598,E2 90.0719} C_DIS
LIN {X -5.5422,Y 3.616,Z 42,A -2.7277,B 0,C 0,E1 0.1598,E2 90.0718} C_DIS
LIN {X -5.9035,Y 2.9934,Z 42,A -2.7673,B 0,C 0,E1 0.1598,E2 90.0717} C_DIS
LIN {X -6.195,Y 2.335,Z 42,A -2.8059,B 0,C 0,E1 0.1598,E2 90.0717} C_DIS
LIN {X -6.4133,Y 1.649,Z 42,A -2.8429,B 0,C 0,E1 0.1598,E2 90.0715} C_DIS
LIN {X -6.5529,Y 0.9427,Z 42,A -2.8779,B 0,C 0,E1 0.1598,E2 90.0715} C_DIS
LIN {X -6.6148,Y 0.2254,Z 42,A -2.9106,B 0,C 0,E1 0.1598,E2 90.0715} C_DIS
LIN {X -6.6032,Y -0.4944,Z 42,A -2.9406,B 0,C 0,E1 0.1598,E2 90.0714} C_DIS
LIN {X -6.5093,Y -1.2082,Z 42,A -2.9674,B 0,C 0,E1 0.1598,E2 90.0714} C_DIS
LIN {X -6.3371,Y -1.9072,Z 42,A -2.9906,B 0,C 0,E1 0.1598,E2 90.0714} C_DIS
LIN {X -6.0949,Y -2.5852,Z 42,A -3.0105,B 0,C 0,E1 0.1598,E2 90.0714} C_DIS
LIN {X -5.7774,Y -3.2314,Z 42,A -3.0262,B 0,C 0,E1 0.1598,E2 90.0714} C_DIS
LIN {X -5.393,Y -3.8401,Z 42,A -3.0379,B 0,C 0,E1 0.1598,E2 90.0714} C_DIS
LIN {X -4.9436,Y -4.4028,Z 42,A -3.0453,B 0,C 0,E1 0.1598,E2 90.0714} C_DIS
LIN {X -4.4363,Y -4.9136,Z 42,A -3.0484,B 0,C 0,E1 0.1598,E2 90.0714} C_DIS
LIN {X -3.8762,Y -5.3659,Z 42,A -3.0471,B 0,C 0,E1 0.1598,E2 90.0714} C_DIS
LIN {X -3.2707,Y -5.755,Z 42,A -3.0414,B 0,C 0,E1 0.1598,E2 90.0714} C_DIS
LIN {X -2.6258,Y -6.0751,Z 42,A -3.0314,B 0,C 0,E1 0.1598,E2 90.0714} C_DIS
LIN {X -1.9504,Y -6.3241,Z 42,A -3.0172,B 0,C 0,E1 0.1598,E2 90.0715} C_DIS
LIN {X -1.2525,Y -6.5009,Z 42,A -2.9991,B 0,C 0,E1 0.1598,E2 90.0715} C_DIS
LIN {X -0.539,Y -6.598,Z 42,A -2.9771,B 0,C 0,E1 0.1598,E2 90.0715} C_DIS
LIN {X -0.539,Y -6.598,Z 42,A -2.9771,B 0,C 0,E1 0.1598,E2 90.0716} C_DIS
Enddeposition()
LIN {X 0,Y -7.5547,Z 42,A -2.9971,B 0,C 0,E1 0.1598,E2 90.0704} C_DIS
Startdeposition()
$VEL.CP = VEL_PRINT
LIN {X -0.9479,Y -7.4978,Z 42,A -3.0305,B 0,C 0,E1 0.1598,E2 90.0715} C_DIS
LIN {X -2.0269,Y -7.2809,Z 42,A -3.0609,B 0,C 0,E1 0.1598,E2 90.0715} C_DIS
LIN {X -2.8839,Y -6.985,Z 42,A -3.0797,B 0,C 0,E1 0.1598,E2 90.0715} C_DIS
LIN {X -3.7192,Y -6.5751,Z 42,A -3.0929,B 0,C 0,E1 0.1598,E2 90.0714} C_DIS
LIN {X -4.3469,Y -6.1752,Z 42,A -3.0989,B 0,C 0,E1 0.1598,E2 90.0714} C_DIS
LIN {X -4.934,Y -5.7178,Z 42,A -3.101,B 0,C 0,E1 0.1598,E2 90.0714} C_DIS
LIN {X -5.6039,Y -5.0722,Z 42,A -3.0981,B 0,C 0,E1 0.1598,E2 90.0712} C_DIS
LIN {X -6.3494,Y -4.0997,Z 42,A -3.0839,B 0,C 0,E1 0.1598,E2 90.0709} C_DIS
LIN {X -6.9165,Y -3.0372,Z 42,A -3.0596,B 0,C 0,E1 0.1598,E2 90.0709} C_DIS
LIN {X -7.1945,Y -2.3121,Z 42,A -3.0393,B 0,C 0,E1 0.1598,E2 90.0711} C_DIS
LIN {X -7.4245,Y -1.3883,Z 42,A -3.0087,B 0,C 0,E1 0.1598,E2 90.0711} C_DIS
LIN {X -7.5441,Y -0.4438,Z 42,A -2.973,B 0,C 0,E1 0.1598,E2 90.0711} C_DIS
LIN {X -7.5208,Y 0.6948,Z 42,A -2.9238,B 0,C 0,E1 0.1598,E2 90.071} C_DIS
LIN {X -7.2909,Y 1.9886,Z 42,A -2.8604,B 0,C 0,E1 0.1598,E2 90.0708} C_DIS
LIN {X -6.7772,Y 3.3426,Z 42,A -2.7841,B 0,C 0,E1 0.1598,E2 90.0708} C_DIS
LIN {X -6.1887,Y 4.3361,Z 42,A -2.7208,B 0,C 0,E1 0.1598,E2 90.0714} C_DIS
LIN {X -5.4823,Y 5.2003,Z 42,A -2.6584,B 0,C 0,E1 0.1598,E2 90.0716} C_DIS
LIN {X -4.6822,Y 5.9317,Z 42,A -2.5981,B 0,C 0,E1 0.1598,E2 90.0718} C_DIS
LIN {X -3.9598,Y 6.4359,Z 42,A -2.5501,B 0,C 0,E1 0.1598,E2 90.072} C_DIS
LIN {X -2.7232,Y 7.0437,Z 42,A -2.4788,B 0,C 0,E1 0.1598,E2 90.0721} C_DIS
LIN {X -1.9987,Y 7.2831,Z 42,A -2.4421,B 0,C 0,E1 0.1598,E2 90.0723} C_DIS
LIN {X -1.2536,Y 7.4478,Z 42,A -2.4076,B 0,C 0,E1 0.1598,E2 90.0723} C_DIS
LIN {X -0.0835,Y 7.557,Z 42,A -2.3598,B 0,C 0,E1 0.1598,E2 90.0724} C_DIS
LIN {X 0.8568,Y 7.5081,Z 42,A -2.3272,B 0,C 0,E1 0.1598,E2 90.0724} C_DIS
LIN {X 1.9792,Y 7.2893,Z 42,A -2.295,B 0,C 0,E1 0.1598,E2 90.0724} C_DIS
LIN {X 2.7809,Y 7.0214,Z 42,A -2.2768,B 0,C 0,E1 0.1598,E2 90.0724} C_DIS
LIN {X 3.7361,Y 6.5692,Z 42,A -2.2607,B 0,C 0,E1 0.1598,E2 90.0724} C_DIS
LIN {X 4.652,Y 5.9505,Z 42,A -2.2531,B 0,C 0,E1 0.1598,E2 90.0724} C_DIS
LIN {X 5.3398,Y 5.3496,Z 42,A -2.2533,B 0,C 0,E1 0.1598,E2 90.0723} C_DIS
LIN {X 6.044,Y 4.5363,Z 42,A -2.2618,B 0,C 0,E1 0.1598,E2 90.0721} C_DIS
LIN {X 6.6656,Y 3.5514,Z 42,A -2.2806,B 0,C 0,E1 0.1598,E2 90.0719} C_DIS
LIN {X 7.0049,Y 2.8263,Z 42,A -2.2993,B 0,C 0,E1 0.1598,E2 90.0722} C_DIS
LIN {X 7.2645,Y 2.0689,Z 42,A -2.322,B 0,C 0,E1 0.1598,E2 90.0722} C_DIS
LIN {X 7.4961,Y 0.9628,Z 42,A -2.3603,B 0,C 0,E1 0.1598,E2 90.0718} C_DIS
LIN {X 7.5586,Y -0.0053,Z 42,A -2.3994,B 0,C 0,E1 0.1598,E2 90.0718} C_DIS
LIN {X 7.5017,Y -0.9134,Z 42,A -2.4404,B 0,C 0,E1 0.1598,E2 90.0718} C_DIS
LIN {X 7.2881,Y -1.9993,Z 42,A -2.4944,B 0,C 0,E1 0.1598,E2 90.0716} C_DIS
LIN {X 6.9122,Y -3.0431,Z 42,A -2.5528,B 0,C 0,E1 0.1598,E2 90.0716} C_DIS
LIN {X 6.5832,Y -3.7043,Z 42,A -2.5934,B 0,C 0,E1 0.1598,E2 90.0719} C_DIS
LIN {X 6.0858,Y -4.482,Z 42,A -2.6448,B 0,C 0,E1 0.1598,E2 90.0717} C_DIS
LIN {X 5.2751,Y -5.4113,Z 42,A -2.7141,B 0,C 0,E1 0.1598,E2 90.0715} C_DIS
LIN {X 4.3948,Y -6.1482,Z 42,A -2.778,B 0,C 0,E1 0.1598,E2 90.0715} C_DIS
LIN {X 3.6808,Y -6.5995,Z 42,A -2.8236,B 0,C 0,E1 0.1598,E2 90.0717} C_DIS
LIN {X 2.7234,Y -7.0499,Z 42,A -2.8779,B 0,C 0,E1 0.1598,E2 90.0717} C_DIS
LIN {X 1.8942,Y -7.3133,Z 42,A -2.9196,B 0,C 0,E1 0.1598,E2 90.0717} C_DIS
LIN {X 1.2131,Y -7.4563,Z 42,A -2.9507,B 0,C 0,E1 0.1598,E2 90.0717} C_DIS
LIN {X 0.5217,Y -7.5347,Z 42,A -2.9793,B 0,C 0,E1 0.1598,E2 90.0717} C_DIS
LIN {X 0.5217,Y -7.5347,Z 42,A -2.9793,B 0,C 0,E1 0.1598,E2 90.0717} C_DIS
Enddeposition()
LIN {X -0.0184,Y -8.4893,Z 42,A -3.0388,B 0,C 0,E1 0.1598,E2 90.0703} C_DIS
Startdeposition()
$VEL.CP = VEL_PRINT
LIN {X 0.9878,Y -8.428,Z 42,A -3.0004,B 0,C 0,E1 0.1598,E2 90.0715} C_DIS
LIN {X 1.7833,Y -8.2958,Z 42,A -2.9657,B 0,C 0,E1 0.1598,E2 90.0716} C_DIS
LIN {X 2.5628,Y -8.0892,Z 42,A -2.9283,B 0,C 0,E1 0.1598,E2 90.0716} C_DIS
LIN {X 3.3193,Y -7.8098,Z 42,A -2.8887,B 0,C 0,E1 0.1598,E2 90.0716} C_DIS
LIN {X 4.046,Y -7.4599,Z 42,A -2.8471,B 0,C 0,E1 0.1598,E2 90.0717} C_DIS
LIN {X 4.7363,Y -7.0427,Z 42,A -2.804,B 0,C 0,E1 0.1598,E2 90.0717} C_DIS
LIN {X 5.646,Y -6.3428,Z 42,A -2.7406,B 0,C 0,E1 0.1598,E2 90.0717} C_DIS
LIN {X 6.3947,Y -5.5852,Z 42,A -2.6807,B 0,C 0,E1 0.1598,E2 90.0717} C_DIS
LIN {X 7.08,Y -4.6787,Z 42,A -2.6167,B 0,C 0,E1 0.1598,E2 90.0717} C_DIS
LIN {X 7.54,Y -3.8947,Z 42,A -2.5664,B 0,C 0,E1 0.1598,E2 90.0718} C_DIS
LIN {X 8.0255,Y -2.7752,Z 42,A -2.5005,B 0,C 0,E1 0.1598,E2 90.0716} C_DIS
LIN {X 8.317,Y -1.7074,Z 42,A -2.4441,B 0,C 0,E1 0.1598,E2 90.0716} C_DIS
LIN {X 8.4472,Y -0.8612,Z 42,A -2.4035,B 0,C 0,E1 0.1598,E2 90.072} C_DIS
LIN {X 8.4797,Y 0.3407,Z 42,A -2.3505,B 0,C 0,E1 0.1598,E2 90.0716} C_DIS
LIN {X 8.4034,Y 1.1857,Z 42,A -2.3177,B 0,C 0,E1 0.1598,E2 90.072} C_DIS
LIN {X 8.2432,Y 2.0189,Z 42,A -2.288,B 0,C 0,E1 0.1598,E2 90.0721} C_DIS
LIN {X 8.0011,Y 2.8321,Z 42,A -2.2623,B 0,C 0,E1 0.1598,E2 90.0721} C_DIS
LIN {X 7.6781,Y 3.6167,Z 42,A -2.2407,B 0,C 0,E1 0.1598,E2 90.0722} C_DIS
LIN {X 7.2787,Y 4.3653,Z 42,A -2.2236,B 0,C 0,E1 0.1598,E2 90.0722} C_DIS
LIN {X 6.8064,Y 5.0702,Z 42,A -2.211,B 0,C 0,E1 0.1598,E2 90.0723} C_DIS
LIN {X 6.2662,Y 5.7245,Z 42,A -2.2031,B 0,C 0,E1 0.1598,E2 90.0723} C_DIS
LIN {X 5.5052,Y 6.4633,Z 42,A -2.1996,B 0,C 0,E1 0.1598,E2 90.0723} C_DIS
LIN {X 4.4698,Y 7.2182,Z 42,A -2.2057,B 0,C 0,E1 0.1598,E2 90.0723} C_DIS
LIN {X 3.5179,Y 7.7237,Z 42,A -2.2195,B 0,C 0,E1 0.1598,E2 90.0724} C_DIS
LIN {X 2.7161,Y 8.0408,Z 42,A -2.2357,B 0,C 0,E1 0.1598,E2 90.0725} C_DIS
LIN {X 1.8862,Y 8.2748,Z 42,A -2.2565,B 0,C 0,E1 0.1598,E2 90.0725} C_DIS
LIN {X 1.037,Y 8.4241,Z 42,A -2.2815,B 0,C 0,E1 0.1598,E2 90.0725} C_DIS
LIN {X 0.177,Y 8.4862,Z 42,A -2.3106,B 0,C 0,E1 0.1598,E2 90.0725} C_DIS
LIN {X -0.6848,Y 8.4593,Z 42,A -2.3436,B 0,C 0,E1 0.1598,E2 90.0725} C_DIS
LIN {X -1.5395,Y 8.3461,Z 42,A -2.38,B 0,C 0,E1 0.1598,E2 90.0724} C_DIS
LIN {X -2.3784,Y 8.1471,Z 42,A -2.4194,B 0,C 0,E1 0.1598,E2 90.0724} C_DIS
LIN {X -3.1929,Y 7.864,Z 42,A -2.4614,B 0,C 0,E1 0.1598,E2 90.0723} C_DIS
LIN {X -3.9743,Y 7.4995,Z 42,A -2.5056,B 0,C 0,E1 0.1598,E2 90.0722} C_DIS
LIN {X -4.7147,Y 7.0576,Z 42,A -2.5516,B 0,C 0,E1 0.1598,E2 90.0721} C_DIS
LIN {X -5.5727,Y 6.4055,Z 42,A -2.6107,B 0,C 0,E1 0.1598,E2 90.0718} C_DIS
LIN {X -6.335,Y 5.6472,Z 42,A -2.6708,B 0,C 0,E1 0.1598,E2 90.0718} C_DIS
LIN {X -6.8985,Y 4.9512,Z 42,A -2.721,B 0,C 0,E1 0.1598,E2 90.0716} C_DIS
LIN {X -7.523,Y 3.9295,Z 42,A -2.7869,B 0,C 0,E1 0.1598,E2 90.0713} C_DIS
LIN {X -7.9859,Y 2.883,Z 42,A -2.8482,B 0,C 0,E1 0.1598,E2 90.0713} C_DIS
LIN {X -8.2906,Y 1.8201,Z 42,A -2.9044,B 0,C 0,E1 0.1598,E2 90.0712} C_DIS
LIN {X -8.4659,Y 0.6516,Z 42,A -2.9601,B 0,C 0,E1 0.1598,E2 90.071} C_DIS
LIN {X -8.4805,Y -0.4338,Z 42,A -3.0066,B 0,C 0,E1 0.1598,E2 90.071} C_DIS
LIN {X -8.3523,Y -1.5025,Z 42,A -3.0471,B 0,C 0,E1 0.1598,E2 90.071} C_DIS
LIN {X -8.1573,Y -2.3411,Z 42,A -3.0756,B 0,C 0,E1 0.1598,E2 90.071} C_DIS
LIN {X -7.8783,Y -3.1557,Z 42,A -3.0999,B 0,C 0,E1 0.1598,E2 90.071} C_DIS
LIN {X -7.518,Y -3.9378,Z 42,A -3.1198,B 0,C 0,E1 0.1598,E2 90.071} C_DIS
LIN {X -7.0804,Y -4.6793,Z 42,A -3.1351,B 0,C 0,E1 0.1598,E2 90.071} C_DIS
LIN {X -6.5697,Y -5.3727,Z 42,A -3.1458,B 0,C 0,E1 0.1598,E2 90.0711} C_DIS
LIN {X -5.9915,Y -6.0108,Z 42,A -3.1517,B 0,C 0,E1 0.1598,E2 90.0711} C_DIS
LIN {X -5.3517,Y -6.5871,Z 42,A -3.1527,B 0,C 0,E1 0.1598,E2 90.0711} C_DIS
LIN {X -4.4767,Y -7.2139,Z 42,A -3.1472,B 0,C 0,E1 0.1598,E2 90.0711} C_DIS
LIN {X -3.388,Y -7.7852,Z 42,A -3.1316,B 0,C 0,E1 0.1598,E2 90.0712} C_DIS
LIN {X -2.3686,Y -8.1491,Z 42,A -3.1098,B 0,C 0,E1 0.1598,E2 90.0714} C_DIS
LIN {X -1.5259,Y -8.3483,Z 42,A -3.0874,B 0,C 0,E1 0.1598,E2 90.0714} C_DIS
LIN {X -0.6674,Y -8.4617,Z 42,A -3.0608,B 0,C 0,E1 0.1598,E2 90.0714} C_DIS
LIN {X -0.6674,Y -8.4617,Z 42,A -3.0608,B 0,C 0,E1 0.1598,E2 90.0714} C_DIS
Enddeposition()
LIN {X 0.0009,Y -4.7544,Z 43,A -2.8639,B 0,C 0,E1 0.1598,E2 90.0604} C_DIS
Startdeposition()
$VEL.CP = VEL_PRINT
LIN {X 0.0009,Y -4.7544,Z 43,A -2.8697,B 0,C 0,E1 0.1598,E2 90.0661} C_DIS
LIN {X -0.8241,Y -4.6794,Z 43,A -2.9017,B 0,C 0,E1 0.1598,E2 90.071} C_DIS
LIN {X -1.4673,Y -4.5192,Z 43,A -2.9191,B 0,C 0,E1 0.1598,E2 90.0716} C_DIS
LIN {X -2.0814,Y -4.2698,Z 43,A -2.931,B 0,C 0,E1 0.1598,E2 90.0716} C_DIS
LIN {X -2.6556,Y -3.9385,Z 43,A -2.938,B 0,C 0,E1 0.1598,E2 90.0716} C_DIS
LIN {X -3.1785,Y -3.5312,Z 43,A -2.9399,B 0,C 0,E1 0.1598,E2 90.0716} C_DIS
LIN {X -3.7414,Y -2.9239,Z 43,A -2.9347,B 0,C 0,E1 0.1598,E2 90.0715} C_DIS
LIN {X -4.0281,Y -2.5179,Z 43,A -2.9281,B 0,C 0,E1 0.1598,E2 90.0715} C_DIS
LIN {X -4.3401,Y -1.9331,Z 43,A -2.9147,B 0,C 0,E1 0.1598,E2 90.0715} C_DIS
LIN {X -4.5661,Y -1.31,Z 43,A -2.8965,B 0,C 0,E1 0.1598,E2 90.0715} C_DIS
LIN {X -4.7045,Y -0.6618,Z 43,A -2.8741,B 0,C 0,E1 0.1598,E2 90.0715} C_DIS
LIN {X -4.7509,Y -0.0007,Z 43,A -2.8478,B 0,C 0,E1 0.1598,E2 90.0715} C_DIS
LIN {X -4.7055,Y 0.6606,Z 43,A -2.8181,B 0,C 0,E1 0.1598,E2 90.0715} C_DIS
LIN {X -4.5677,Y 1.309,Z 43,A -2.7855,B 0,C 0,E1 0.1598,E2 90.0716} C_DIS
LIN {X -4.3406,Y 1.9317,Z 43,A -2.7508,B 0,C 0,E1 0.1598,E2 90.0717} C_DIS
LIN {X -4.0304,Y 2.5174,Z 43,A -2.7146,B 0,C 0,E1 0.1598,E2 90.0717} C_DIS
LIN {X -3.6402,Y 3.0534,Z 43,A -2.6776,B 0,C 0,E1 0.1598,E2 90.0719} C_DIS
LIN {X -3.1804,Y 3.531,Z 43,A -2.6404,B 0,C 0,E1 0.1598,E2 90.0719} C_DIS
LIN {X -2.658,Y 3.9393,Z 43,A -2.6039,B 0,C 0,E1 0.1598,E2 90.072} C_DIS
LIN {X -2.0842,Y 4.2716,Z 43,A -2.5687,B 0,C 0,E1 0.1598,E2 90.072} C_DIS
LIN {X -1.4695,Y 4.5202,Z 43,A -2.5355,B 0,C 0,E1 0.1598,E2 90.0722} C_DIS
LIN {X -0.8262,Y 4.6807,Z 43,A -2.505,B 0,C 0,E1 0.1598,E2 90.0722} C_DIS
LIN {X -0.1668,Y 4.7489,Z 43,A -2.4778,B 0,C 0,E1 0.1598,E2 90.0722} C_DIS
LIN {X 0.4958,Y 4.7261,Z 43,A -2.4544,B 0,C 0,E1 0.1598,E2 90.0722} C_DIS
LIN {X 1.1485,Y 4.6103,Z 43,A -2.4352,B 0,C 0,E1 0.1598,E2 90.0723} C_DIS
LIN {X 1.7791,Y 4.4061,Z 43,A -2.4206,B 0,C 0,E1 0.1598,E2 90.0723} C_DIS
LIN {X 2.3741,Y 4.1139,Z 43,A -2.4111,B 0,C 0,E1 0.1598,E2 90.0723} C_DIS
LIN {X 3.0517,Y 3.6382,Z 43,A -2.4063,B 0,C 0,E1 0.1598,E2 90.0723} C_DIS
LIN {X 3.6907,Y 2.9897,Z 43,A -2.4102,B 0,C 0,E1 0.1598,E2 90.0721} C_DIS
LIN {X 4.0289,Y 2.5184,Z 43,A -2.4179,B 0,C 0,E1 0.1598,E2 90.0721} C_DIS
LIN {X 4.3716,Y 1.8563,Z 43,A -2.4333,B 0,C 0,E1 0.1598,E2 90.0721} C_DIS
LIN {X 4.5664,Y 1.31,Z 43,A -2.4495,B 0,C 0,E1 0.1598,E2 90.0721} C_DIS
LIN {X 4.7043,Y 0.6618,Z 43,A -2.472,B 0,C 0,E1 0.1598,E2 90.0721} C_DIS
LIN {X 4.7509,Y 0.0006,Z 43,A -2.4984,B 0,C 0,E1 0.1598,E2 90.072} C_DIS
LIN {X 4.7055,Y -0.6607,Z 43,A -2.5283,B 0,C 0,E1 0.1598,E2 90.072} C_DIS
LIN {X 4.5677,Y -1.3091,Z 43,A -2.561,B 0,C 0,E1 0.1598,E2 90.072} C_DIS
LIN {X 4.3406,Y -1.9318,Z 43,A -2.5959,B 0,C 0,E1 0.1598,E2 90.072} C_DIS
LIN {X 4.0307,Y -2.5177,Z 43,A -2.6323,B 0,C 0,E1 0.1598,E2 90.0719} C_DIS
LIN {X 3.6413,Y -3.0545,Z 43,A -2.6695,B 0,C 0,E1 0.1598,E2 90.0719} C_DIS
LIN {X 3.1804,Y -3.5311,Z 43,A -2.7067,B 0,C 0,E1 0.1598,E2 90.0719} C_DIS
LIN {X 2.6582,Y -3.9396,Z 43,A -2.7434,B 0,C 0,E1 0.1598,E2 90.0719} C_DIS
LIN {X 2.084,Y -4.2713,Z 43,A -2.7786,B 0,C 0,E1 0.1598,E2 90.0719} C_DIS
LIN {X 1.4695,Y -4.5201,Z 43,A -2.8118,B 0,C 0,E1 0.1598,E2 90.0718} C_DIS
LIN {X 0.8262,Y -4.6808,Z 43,A -2.8422,B 0,C 0,E1 0.1598,E2 90.0718} C_DIS
LIN {X 0.0009,Y -4.7544,Z 43,A -2.8757,B 0,C 0,E1 0.1598,E2 90.0718} C_DIS
Enddeposition()
LIN {X 0.0009,Y -4.7544,Z 43,A -2.8757,B 0,C 0,E1 0.1598,E2 90.0718} C_DIS
Startdeposition()
$VEL.CP = VEL_PRINT
LIN {X 0.2414,Y -5.6798,Z 43,A -2.9058,B 0,C 0,E1 0.1598,E2 90.0711} C_DIS
LIN {X 1.0535,Y -5.5875,Z 43,A -2.8726,B 0,C 0,E1 0.1598,E2 90.0717} C_DIS
LIN {X 1.843,Y -5.3766,Z 43,A -2.8347,B 0,C 0,E1 0.1598,E2 90.0717} C_DIS
LIN {X 2.5956,Y -5.0582,Z 43,A -2.7934,B 0,C 0,E1 0.1598,E2 90.0718} C_DIS
LIN {X 3.2941,Y -4.6339,Z 43,A -2.7497,B 0,C 0,E1 0.1598,E2 90.0718} C_DIS
LIN {X 3.9246,Y -4.1138,Z 43,A -2.7043,B 0,C 0,E1 0.1598,E2 90.0718} C_DIS
LIN {X 4.4714,Y -3.5068,Z 43,A -2.6583,B 0,C 0,E1 0.1598,E2 90.0718} C_DIS
LIN {X 4.9276,Y -2.8291,Z 43,A -2.6126,B 0,C 0,E1 0.1598,E2 90.0718} C_DIS
LIN {X 5.2839,Y -2.094,Z 43,A -2.5681,B 0,C 0,E1 0.1598,E2 90.0718} C_DIS
LIN {X 5.5302,Y -1.3148,Z 43,A -2.5258,B 0,C 0,E1 0.1598,E2 90.0718} C_DIS
LIN {X 5.6633,Y -0.5084,Z 43,A -2.4865,B 0,C 0,E1 0.1598,E2 90.0718} C_DIS
LIN {X 5.6766,Y 0.3088,Z 43,A -2.4511,B 0,C 0,E1 0.1598,E2 90.0719} C_DIS
LIN {X 5.5735,Y 1.1194,Z 43,A -2.4204,B 0,C 0,E1 0.1598,E2 90.0719} C_DIS
LIN {X 5.3559,Y 1.9072,Z 43,A -2.3948,B 0,C 0,E1 0.1598,E2 90.072} C_DIS
LIN {X 5.0264,Y 2.6551,Z 43,A -2.3751,B 0,C 0,E1 0.1598,E2 90.072} C_DIS
LIN {X 4.5929,Y 3.3478,Z 43,A -2.3617,B 0,C 0,E1 0.1598,E2 90.0721} C_DIS
LIN {X 4.0651,Y 3.9713,Z 43,A -2.3546,B 0,C 0,E1 0.1598,E2 90.0721} C_DIS
LIN {X 3.4531,Y 4.5125,Z 43,A -2.3542,B 0,C 0,E1 0.1598,E2 90.0722} C_DIS
LIN {X 2.7706,Y 4.9615,Z 43,A -2.3603,B 0,C 0,E1 0.1598,E2 90.0722} C_DIS
LIN {X 2.0306,Y 5.3074,Z 43,A -2.373,B 0,C 0,E1 0.1598,E2 90.0723} C_DIS
LIN {X 1.2485,Y 5.5435,Z 43,A -2.3918,B 0,C 0,E1 0.1598,E2 90.0723} C_DIS
LIN {X 0.4407,Y 5.6652,Z 43,A -2.4164,B 0,C 0,E1 0.1598,E2 90.0723} C_DIS
LIN {X -0.3761,Y 5.6696,Z 43,A -2.4464,B 0,C 0,E1 0.1598,E2 90.0723} C_DIS
LIN {X -1.1854,Y 5.5581,Z 43,A -2.481,B 0,C 0,E1 0.1598,E2 90.0723} C_DIS
LIN {X -1.9696,Y 5.3296,Z 43,A -2.5195,B 0,C 0,E1 0.1598,E2 90.0722} C_DIS
LIN {X -2.7139,Y 4.9929,Z 43,A -2.5612,B 0,C 0,E1 0.1598,E2 90.0722} C_DIS
LIN {X -3.4019,Y 4.5523,Z 43,A -2.6052,B 0,C 0,E1 0.1598,E2 90.072} C_DIS
LIN {X -4.0205,Y 4.0184,Z 43,A -2.6506,B 0,C 0,E1 0.1598,E2 90.0719} C_DIS
LIN {X -4.5543,Y 3.3998,Z 43,A -2.6964,B 0,C 0,E1 0.1598,E2 90.0718} C_DIS
LIN {X -4.9962,Y 2.7124,Z 43,A -2.7417,B 0,C 0,E1 0.1598,E2 90.0717} C_DIS
LIN {X -5.3323,Y 1.9676,Z 43,A -2.7856,B 0,C 0,E1 0.1598,E2 90.0716} C_DIS
LIN {X -5.5591,Y 1.1826,Z 43,A -2.8271,B 0,C 0,E1 0.1598,E2 90.0715} C_DIS
LIN {X -5.6716,Y 0.3734,Z 43,A -2.8655,B 0,C 0,E1 0.1598,E2 90.0715} C_DIS
LIN {X -5.6676,Y -0.4437,Z 43,A -2.9,B 0,C 0,E1 0.1598,E2 90.0714} C_DIS
LIN {X -5.5449,Y -1.2517,Z 43,A -2.9297,B 0,C 0,E1 0.1598,E2 90.0714} C_DIS
LIN {X -5.3082,Y -2.0338,Z 43,A -2.9542,B 0,C 0,E1 0.1598,E2 90.0714} C_DIS
LIN {X -4.8629,Y -2.9531,Z 43,A -2.9766,B 0,C 0,E1 0.1598,E2 90.0711} C_DIS
LIN {X -4.0762,Y -3.9694,Z 43,A -2.9908,B 0,C 0,E1 0.1598,E2 90.0711} C_DIS
LIN {X -3.3533,Y -4.5902,Z 43,A -2.9909,B 0,C 0,E1 0.1598,E2 90.0714} C_DIS
LIN {X -2.7083,Y -4.9965,Z 43,A -2.9846,B 0,C 0,E1 0.1598,E2 90.0714} C_DIS
LIN {X -2.0153,Y -5.3136,Z 43,A -2.9727,B 0,C 0,E1 0.1598,E2 90.0716} C_DIS
LIN {X -1.2865,Y -5.5358,Z 43,A -2.9554,B 0,C 0,E1 0.1598,E2 90.0716} C_DIS
LIN {X -0.5342,Y -5.658,Z 43,A -2.9331,B 0,C 0,E1 0.1598,E2 90.0716} C_DIS
LIN {X -0.5342,Y -5.658,Z 43,A -2.9331,B 0,C 0,E1 0.1598,E2 90.0716} C_DIS
Enddeposition()
LIN {X 0.0755,Y -6.6226,Z 43,A -2.9507,B 0,C 0,E1 0.1598,E2 90.0704} C_DIS
Startdeposition()
$VEL.CP = VEL_PRINT
LIN {X -0.7997,Y -6.571,Z 43,A -2.9817,B 0,C 0,E1 0.1598,E2 90.0715} C_DIS
LIN {X -1.4906,Y -6.4509,Z 43,A -3.002,B 0,C 0,E1 0.1598,E2 90.0715} C_DIS
LIN {X -2.1646,Y -6.2567,Z 43,A -3.0185,B 0,C 0,E1 0.1598,E2 90.0715} C_DIS
LIN {X -2.8144,Y -5.9923,Z 43,A -3.031,B 0,C 0,E1 0.1598,E2 90.0715} C_DIS
LIN {X -3.4331,Y -5.6618,Z 43,A -3.0397,B 0,C 0,E1 0.1598,E2 90.0715} C_DIS
LIN {X -4.0127,Y -5.2666,Z 43,A -3.0441,B 0,C 0,E1 0.1598,E2 90.0715} C_DIS
LIN {X -4.5481,Y -4.8134,Z 43,A -3.0445,B 0,C 0,E1 0.1598,E2 90.0714} C_DIS
LIN {X -5.0304,Y -4.3042,Z 43,A -3.0406,B 0,C 0,E1 0.1598,E2 90.0714} C_DIS
LIN {X -5.457,Y -3.7473,Z 43,A -3.0326,B 0,C 0,E1 0.1598,E2 90.0714} C_DIS
LIN {X -5.822,Y -3.1484,Z 43,A -3.0206,B 0,C 0,E1 0.1598,E2 90.0714} C_DIS
LIN {X -6.124,Y -2.5154,Z 43,A -3.0048,B 0,C 0,E1 0.1598,E2 90.0714} C_DIS
LIN {X -6.3541,Y -1.8527,Z 43,A -2.9852,B 0,C 0,E1 0.1598,E2 90.0714} C_DIS
LIN {X -6.515,Y -1.1702,Z 43,A -2.9622,B 0,C 0,E1 0.1598,E2 90.0714} C_DIS
LIN {X -6.6034,Y -0.4743,Z 43,A -2.936,B 0,C 0,E1 0.1598,E2 90.0714} C_DIS
LIN {X -6.6151,Y 0.227,Z 43,A -2.9067,B 0,C 0,E1 0.1598,E2 90.0714} C_DIS
LIN {X -6.5549,Y 0.9257,Z 43,A -2.8749,B 0,C 0,E1 0.1598,E2 90.0714} C_DIS
LIN {X -6.4186,Y 1.6137,Z 43,A -2.8408,B 0,C 0,E1 0.1598,E2 90.0715} C_DIS
LIN {X -6.2122,Y 2.284,Z 43,A -2.8048,B 0,C 0,E1 0.1598,E2 90.0715} C_DIS
LIN {X -5.9355,Y 2.9284,Z 43,A -2.7674,B 0,C 0,E1 0.1598,E2 90.0717} C_DIS
LIN {X -5.5928,Y 3.5403,Z 43,A -2.7289,B 0,C 0,E1 0.1598,E2 90.0717} C_DIS
LIN {X -5.1873,Y 4.1126,Z 43,A -2.6897,B 0,C 0,E1 0.1598,E2 90.0718} C_DIS
LIN {X -4.7232,Y 4.6383,Z 43,A -2.6504,B 0,C 0,E1 0.1598,E2 90.0718} C_DIS
LIN {X -4.2054,Y 5.1114,Z 43,A -2.6113,B 0,C 0,E1 0.1598,E2 90.072} C_DIS
LIN {X -3.641,Y 5.5279,Z 43,A -2.5729,B 0,C 0,E1 0.1598,E2 90.072} C_DIS
LIN {X -3.036,Y 5.8827,Z 43,A -2.5356,B 0,C 0,E1 0.1598,E2 90.0721} C_DIS
LIN {X -2.2332,Y 6.2353,Z 43,A -2.491,B 0,C 0,E1 0.1598,E2 90.0721} C_DIS
LIN {X -1.2406,Y 6.5014,Z 43,A -2.4431,B 0,C 0,E1 0.1598,E2 90.0723} C_DIS
LIN {X -0.5555,Y 6.5957,Z 43,A -2.4139,B 0,C 0,E1 0.1598,E2 90.0723} C_DIS
LIN {X 0.1358,Y 6.6193,Z 43,A -2.3874,B 0,C 0,E1 0.1598,E2 90.0723} C_DIS
LIN {X 0.8257,Y 6.5687,Z 43,A -2.3641,B 0,C 0,E1 0.1598,E2 90.0724} C_DIS
LIN {X 1.5064,Y 6.4466,Z 43,A -2.3441,B 0,C 0,E1 0.1598,E2 90.0724} C_DIS
LIN {X 2.1709,Y 6.2545,Z 43,A -2.3278,B 0,C 0,E1 0.1598,E2 90.0724} C_DIS
LIN {X 2.8115,Y 5.9934,Z 43,A -2.3152,B 0,C 0,E1 0.1598,E2 90.0724} C_DIS
LIN {X 3.4215,Y 5.6672,Z 43,A -2.3066,B 0,C 0,E1 0.1598,E2 90.0724} C_DIS
LIN {X 3.9948,Y 5.2801,Z 43,A -2.3019,B 0,C 0,E1 0.1598,E2 90.0724} C_DIS
LIN {X 4.5232,Y 4.8337,Z 43,A -2.3013,B 0,C 0,E1 0.1598,E2 90.0724} C_DIS
LIN {X 5.0032,Y 4.3357,Z 43,A -2.3048,B 0,C 0,E1 0.1598,E2 90.0724} C_DIS
LIN {X 5.4271,Y 3.7891,Z 43,A -2.3124,B 0,C 0,E1 0.1598,E2 90.0724} C_DIS
LIN {X 5.7957,Y 3.2037,Z 43,A -2.3238,B 0,C 0,E1 0.1598,E2 90.0723} C_DIS
LIN {X 6.0986,Y 2.5817,Z 43,A -2.3391,B 0,C 0,E1 0.1598,E2 90.0723} C_DIS
LIN {X 6.3339,Y 1.9312,Z 43,A -2.3581,B 0,C 0,E1 0.1598,E2 90.0722} C_DIS
LIN {X 6.4986,Y 1.2594,Z 43,A -2.3807,B 0,C 0,E1 0.1598,E2 90.0722} C_DIS
LIN {X 6.5961,Y 0.5747,Z 43,A -2.4063,B 0,C 0,E1 0.1598,E2 90.0721} C_DIS
LIN {X 6.6174,Y -0.1166,Z 43,A -2.435,B 0,C 0,E1 0.1598,E2 90.0721} C_DIS
LIN {X 6.5706,Y -0.8066,Z 43,A -2.4661,B 0,C 0,E1 0.1598,E2 90.0721} C_DIS
LIN {X 6.4495,Y -1.4876,Z 43,A -2.4996,B 0,C 0,E1 0.1598,E2 90.072} C_DIS
LIN {X 6.2609,Y -2.153,Z 43,A -2.535,B 0,C 0,E1 0.1598,E2 90.072} C_DIS
LIN {X 6.0017,Y -2.7943,Z 43,A -2.5719,B 0,C 0,E1 0.1598,E2 90.072} C_DIS
LIN {X 5.6779,Y -3.4056,Z 43,A -2.6099,B 0,C 0,E1 0.1598,E2 90.0719} C_DIS
LIN {X 5.2905,Y -3.9788,Z 43,A -2.6486,B 0,C 0,E1 0.1598,E2 90.0719} C_DIS
LIN {X 4.8477,Y -4.5102,Z 43,A -2.6875,B 0,C 0,E1 0.1598,E2 90.0719} C_DIS
LIN {X 4.3508,Y -4.9914,Z 43,A -2.7263,B 0,C 0,E1 0.1598,E2 90.0719} C_DIS
LIN {X 3.8062,Y -5.4178,Z 43,A -2.7645,B 0,C 0,E1 0.1598,E2 90.0718} C_DIS
LIN {X 3.2198,Y -5.7847,Z 43,A -2.8017,B 0,C 0,E1 0.1598,E2 90.0718} C_DIS
LIN {X 2.5994,Y -6.0909,Z 43,A -2.8375,B 0,C 0,E1 0.1598,E2 90.0718} C_DIS
LIN {X 1.9498,Y -6.3286,Z 43,A -2.8715,B 0,C 0,E1 0.1598,E2 90.0718} C_DIS
LIN {X 1.2783,Y -6.4949,Z 43,A -2.9032,B 0,C 0,E1 0.1598,E2 90.0717} C_DIS
LIN {X 0.5937,Y -6.5927,Z 43,A -2.9325,B 0,C 0,E1 0.1598,E2 90.0717} C_DIS
LIN {X 0.5937,Y -6.5927,Z 43,A -2.9325,B 0,C 0,E1 0.1598,E2 90.0717} C_DIS
Enddeposition()
LIN {X 0.0972,Y -7.5523,Z 43,A -2.9905,B 0,C 0,E1 0.1598,E2 90.0704} C_DIS
Startdeposition()
$VEL.CP = VEL_PRINT
LIN {X 0.8488,Y -7.509,Z 43,A -2.9623,B 0,C 0,E1 0.1598,E2 90.0716} C_DIS
LIN {X 1.9653,Y -7.2969,Z 43,A -2.9123,B 0,C 0,E1 0.1598,E2 90.0716} C_DIS
LIN {X 3.0511,Y -6.9099,Z 43,A -2.856,B 0,C 0,E1 0.1598,E2 90.0716} C_DIS
LIN {X 3.963,Y -6.4339,Z 43,A -2.8022,B 0,C 0,E1 0.1598,E2 90.0717} C_DIS
LIN {X 4.8742,Y -5.7714,Z 43,A -2.7404,B 0,C 0,E1 0.1598,E2 90.0717} C_DIS
LIN {X 5.4534,Y -5.2269,Z 43,A -2.696,B 0,C 0,E1 0.1598,E2 90.0718} C_DIS
LIN {X 5.9727,Y -4.6248,Z 43,A -2.6512,B 0,C 0,E1 0.1598,E2 90.0718} C_DIS
LIN {X 6.532,Y -3.8033,Z 43,A -2.5954,B 0,C 0,E1 0.1598,E2 90.0717} C_DIS
LIN {X 6.9801,Y -2.8868,Z 43,A -2.5397,B 0,C 0,E1 0.1598,E2 90.0717} C_DIS
LIN {X 7.3029,Y -1.9424,Z 43,A -2.4875,B 0,C 0,E1 0.1598,E2 90.0717} C_DIS
LIN {X 7.4865,Y -1.0406,Z 43,A -2.4423,B 0,C 0,E1 0.1598,E2 90.0719} C_DIS
LIN {X 7.5522,Y 0.1553,Z 43,A -2.3884,B 0,C 0,E1 0.1598,E2 90.0715} C_DIS
LIN {X 7.4458,Y 1.2938,Z 43,A -2.3437,B 0,C 0,E1 0.1598,E2 90.0715} C_DIS
LIN {X 7.1901,Y 2.3262,Z 43,A -2.3094,B 0,C 0,E1 0.1598,E2 90.0719} C_DIS
LIN {X 6.7351,Y 3.4196,Z 43,A -2.2794,B 0,C 0,E1 0.1598,E2 90.0719} C_DIS
LIN {X 6.3197,Y 4.1349,Z 43,A -2.2646,B 0,C 0,E1 0.1598,E2 90.0722} C_DIS
LIN {X 5.6992,Y 4.9621,Z 43,A -2.2521,B 0,C 0,E1 0.1598,E2 90.0721} C_DIS
LIN {X 4.8915,Y 5.7549,Z 43,A -2.2482,B 0,C 0,E1 0.1598,E2 90.0721} C_DIS
LIN {X 4.0938,Y 6.3531,Z 43,A -2.2523,B 0,C 0,E1 0.1598,E2 90.0723} C_DIS
LIN {X 2.9185,Y 6.9703,Z 43,A -2.2695,B 0,C 0,E1 0.1598,E2 90.0723} C_DIS
LIN {X 2.2094,Y 7.2266,Z 43,A -2.2849,B 0,C 0,E1 0.1598,E2 90.0725} C_DIS
LIN {X 0.9647,Y 7.4959,Z 43,A -2.3195,B 0,C 0,E1 0.1598,E2 90.0725} C_DIS
LIN {X 0.1456,Y 7.5556,Z 43,A -2.3472,B 0,C 0,E1 0.1598,E2 90.0725} C_DIS
LIN {X -0.9816,Y 7.4898,Z 43,A -2.3916,B 0,C 0,E1 0.1598,E2 90.0724} C_DIS
LIN {X -1.9392,Y 7.3037,Z 43,A -2.4348,B 0,C 0,E1 0.1598,E2 90.0724} C_DIS
LIN {X -3.1982,Y 6.8473,Z 43,A -2.5005,B 0,C 0,E1 0.1598,E2 90.0721} C_DIS
LIN {X -4.1759,Y 6.2969,Z 43,A -2.5598,B 0,C 0,E1 0.1598,E2 90.0721} C_DIS
LIN {X -4.9973,Y 5.6691,Z 43,A -2.6166,B 0,C 0,E1 0.1598,E2 90.0719} C_DIS
LIN {X -5.6857,Y 4.9694,Z 43,A -2.6716,B 0,C 0,E1 0.1598,E2 90.0718} C_DIS
LIN {X -6.3868,Y 4.0392,Z 43,A -2.7366,B 0,C 0,E1 0.1598,E2 90.0715} C_DIS
LIN {X -6.7795,Y 3.3377,Z 43,A -2.7809,B 0,C 0,E1 0.1598,E2 90.0716} C_DIS
LIN {X -7.1906,Y 2.3244,Z 43,A -2.8386,B 0,C 0,E1 0.1598,E2 90.0713} C_DIS
LIN {X -7.4374,Y 1.3135,Z 43,A -2.8905,B 0,C 0,E1 0.1598,E2 90.0713} C_DIS
LIN {X -7.5386,Y 0.4873,Z 43,A -2.9293,B 0,C 0,E1 0.1598,E2 90.0713} C_DIS
LIN {X -7.5368,Y -0.5533,Z 43,A -2.973,B 0,C 0,E1 0.1598,E2 90.071} C_DIS
LIN {X -7.3776,Y -1.6245,Z 43,A -3.0125,B 0,C 0,E1 0.1598,E2 90.071} C_DIS
LIN {X -7.1198,Y -2.533,Z 43,A -3.0416,B 0,C 0,E1 0.1598,E2 90.071} C_DIS
LIN {X -6.722,Y -3.4561,Z 43,A -3.0662,B 0,C 0,E1 0.1598,E2 90.071} C_DIS
LIN {X -6.1316,Y -4.4104,Z 43,A -3.0849,B 0,C 0,E1 0.1598,E2 90.071} C_DIS
LIN {X -5.6762,Y -4.9822,Z 43,A -3.0927,B 0,C 0,E1 0.1598,E2 90.0713} C_DIS
LIN {X -5.1684,Y -5.5079,Z 43,A -3.0964,B 0,C 0,E1 0.1598,E2 90.0713} C_DIS
LIN {X -4.6107,Y -5.9803,Z 43,A -3.096,B 0,C 0,E1 0.1598,E2 90.0713} C_DIS
LIN {X -3.4991,Y -6.6994,Z 43,A -3.0856,B 0,C 0,E1 0.1598,E2 90.0711} C_DIS
LIN {X -2.1252,Y -7.2477,Z 43,A -3.0586,B 0,C 0,E1 0.1598,E2 90.0713} C_DIS
LIN {X -1.0078,Y -7.491,Z 43,A -3.0282,B 0,C 0,E1 0.1598,E2 90.0715} C_DIS
LIN {X 0.0972,Y -7.5523,Z 43,A -2.9903,B 0,C 0,E1 0.1598,E2 90.0715} C_DIS
Enddeposition()
LIN {X 0.0972,Y -7.5523,Z 43,A -2.9903,B 0,C 0,E1 0.1598,E2 90.0715} C_DIS
Startdeposition()
$VEL.CP = VEL_PRINT
LIN {X -0.4592,Y -8.474,Z 43,A -3.0496,B 0,C 0,E1 0.1598,E2 90.0709} C_DIS
LIN {X -1.2386,Y -8.3952,Z 43,A -3.0753,B 0,C 0,E1 0.1598,E2 90.0714} C_DIS
LIN {X -2.0075,Y -8.2451,Z 43,A -3.0971,B 0,C 0,E1 0.1598,E2 90.0714} C_DIS
LIN {X -3.1687,Y -7.8785,Z 43,A -3.124,B 0,C 0,E1 0.1598,E2 90.0714} C_DIS
LIN {X -4.2675,Y -7.3364,Z 43,A -3.1412,B 0,C 0,E1 0.1598,E2 90.0712} C_DIS
LIN {X -4.9766,Y -6.8748,Z 43,A -3.1476,B 0,C 0,E1 0.1598,E2 90.0712} C_DIS
LIN {X -5.6362,Y -6.345,Z 43,A -3.1493,B 0,C 0,E1 0.1598,E2 90.0712} C_DIS
LIN {X -6.2395,Y -5.7518,Z 43,A -3.1462,B 0,C 0,E1 0.1598,E2 90.0712} C_DIS
LIN {X -6.7812,Y -5.102,Z 43,A -3.1385,B 0,C 0,E1 0.1598,E2 90.0712} C_DIS
LIN {X -7.2555,Y -4.4015,Z 43,A -3.1262,B 0,C 0,E1 0.1598,E2 90.0712} C_DIS
LIN {X -7.657,Y -3.6569,Z 43,A -3.1094,B 0,C 0,E1 0.1598,E2 90.0712} C_DIS
LIN {X -7.9837,Y -2.8766,Z 43,A -3.0883,B 0,C 0,E1 0.1598,E2 90.0712} C_DIS
LIN {X -8.2302,Y -2.0674,Z 43,A -3.0631,B 0,C 0,E1 0.1598,E2 90.0712} C_DIS
LIN {X -8.395,Y -1.2377,Z 43,A -3.034,B 0,C 0,E1 0.1598,E2 90.0712} C_DIS
LIN {X -8.4767,Y -0.3957,Z 43,A -3.0014,B 0,C 0,E1 0.1598,E2 90.0712} C_DIS
LIN {X -8.4578,Y 0.7642,Z 43,A -2.9513,B 0,C 0,E1 0.1598,E2 90.071} C_DIS
LIN {X -8.2526,Y 2.0002,Z 43,A -2.8912,B 0,C 0,E1 0.1598,E2 90.0708} C_DIS
LIN {X -7.8756,Y 3.1618,Z 43,A -2.8284,B 0,C 0,E1 0.1598,E2 90.071} C_DIS
LIN {X -7.5013,Y 3.9688,Z 43,A -2.7809,B 0,C 0,E1 0.1598,E2 90.0715} C_DIS
LIN {X -7.0449,Y 4.7324,Z 43,A -2.7318,B 0,C 0,E1 0.1598,E2 90.0716} C_DIS
LIN {X -6.2616,Y 5.7354,Z 43,A -2.6604,B 0,C 0,E1 0.1598,E2 90.0716} C_DIS
LIN {X -5.4655,Y 6.4927,Z 43,A -2.5992,B 0,C 0,E1 0.1598,E2 90.0718} C_DIS
LIN {X -4.7647,Y 7.0233,Z 43,A -2.551,B 0,C 0,E1 0.1598,E2 90.072} C_DIS
LIN {X -4.0128,Y 7.4787,Z 43,A -2.504,B 0,C 0,E1 0.1598,E2 90.0721} C_DIS
LIN {X -3.2179,Y 7.854,Z 43,A -2.4588,B 0,C 0,E1 0.1598,E2 90.0722} C_DIS
LIN {X -2.3882,Y 8.1445,Z 43,A -2.4159,B 0,C 0,E1 0.1598,E2 90.0723} C_DIS
LIN {X -1.2229,Y 8.4028,Z 43,A -2.362,B 0,C 0,E1 0.1598,E2 90.0723} C_DIS
LIN {X 0.0282,Y 8.487,Z 43,A -2.3122,B 0,C 0,E1 0.1598,E2 90.0725} C_DIS
LIN {X 0.9179,Y 8.4373,Z 43,A -2.2815,B 0,C 0,E1 0.1598,E2 90.0725} C_DIS
LIN {X 1.7972,Y 8.294,Z 43,A -2.2551,B 0,C 0,E1 0.1598,E2 90.0725} C_DIS
LIN {X 2.6568,Y 8.0593,Z 43,A -2.2333,B 0,C 0,E1 0.1598,E2 90.0725} C_DIS
LIN {X 3.4873,Y 7.7366,Z 43,A -2.2163,B 0,C 0,E1 0.1598,E2 90.0725} C_DIS
LIN {X 4.4723,Y 7.2166,Z 43,A -2.2019,B 0,C 0,E1 0.1598,E2 90.0725} C_DIS
LIN {X 5.508,Y 6.4608,Z 43,A -2.1957,B 0,C 0,E1 0.1598,E2 90.0723} C_DIS
LIN {X 6.2864,Y 5.7016,Z 43,A -2.1993,B 0,C 0,E1 0.1598,E2 90.0723} C_DIS
LIN {X 7.0847,Y 4.6818,Z 43,A -2.2131,B 0,C 0,E1 0.1598,E2 90.072} C_DIS
LIN {X 7.6089,Y 3.7671,Z 43,A -2.2328,B 0,C 0,E1 0.1598,E2 90.072} C_DIS
LIN {X 7.989,Y 2.8746,Z 43,A -2.257,B 0,C 0,E1 0.1598,E2 90.0721} C_DIS
LIN {X 8.2818,Y 1.875,Z 43,A -2.2887,B 0,C 0,E1 0.1598,E2 90.072} C_DIS
LIN {X 8.4548,Y 0.7397,Z 43,A -2.3306,B 0,C 0,E1 0.1598,E2 90.0717} C_DIS
LIN {X 8.4858,Y -0.3103,Z 43,A -2.3743,B 0,C 0,E1 0.1598,E2 90.0717} C_DIS
LIN {X 8.4196,Y -1.1042,Z 43,A -2.411,B 0,C 0,E1 0.1598,E2 90.072} C_DIS
LIN {X 8.1659,Y -2.3143,Z 43,A -2.4716,B 0,C 0,E1 0.1598,E2 90.0715} C_DIS
LIN {X 7.895,Y -3.1146,Z 43,A -2.5161,B 0,C 0,E1 0.1598,E2 90.0718} C_DIS
LIN {X 7.546,Y -3.884,Z 43,A -2.5618,B 0,C 0,E1 0.1598,E2 90.0718} C_DIS
LIN {X 7.1222,Y -4.6148,Z 43,A -2.6086,B 0,C 0,E1 0.1598,E2 90.0718} C_DIS
LIN {X 6.628,Y -5.2999,Z 43,A -2.6561,B 0,C 0,E1 0.1598,E2 90.0718} C_DIS
LIN {X 6.0681,Y -5.9325,Z 43,A -2.7037,B 0,C 0,E1 0.1598,E2 90.0718} C_DIS
LIN {X 5.4481,Y -6.5064,Z 43,A -2.7509,B 0,C 0,E1 0.1598,E2 90.0718} C_DIS
LIN {X 4.7743,Y -7.0158,Z 43,A -2.7974,B 0,C 0,E1 0.1598,E2 90.0718} C_DIS
LIN {X 4.0531,Y -7.4556,Z 43,A -2.8427,B 0,C 0,E1 0.1598,E2 90.0717} C_DIS
LIN {X 3.0983,Y -7.9067,Z 43,A -2.8969,B 0,C 0,E1 0.1598,E2 90.0717} C_DIS
LIN {X 1.9757,Y -8.2542,Z 43,A -2.9529,B 0,C 0,E1 0.1598,E2 90.0716} C_DIS
LIN {X 1.1611,Y -8.4072,Z 43,A -2.9893,B 0,C 0,E1 0.1598,E2 90.0716} C_DIS
LIN {X 0.1284,Y -8.489,Z 43,A -3.0306,B 0,C 0,E1 0.1598,E2 90.0716} C_DIS
Enddeposition()
LIN {X 0.0009,Y -4.7544,Z 44,A -2.8617,B 0,C 0,E1 0.1598,E2 90.0604} C_DIS
Startdeposition()
$VEL.CP = VEL_PRINT
LIN {X 0.0009,Y -4.7544,Z 44,A -2.8674,B 0,C 0,E1 0.1598,E2 90.0661} C_DIS
LIN {X 0.8444,Y -4.6754,Z 44,A -2.8381,B 0,C 0,E1 0.1598,E2 90.0711} C_DIS
LIN {X 1.5011,Y -4.5075,Z 44,A -2.8074,B 0,C 0,E1 0.1598,E2 90.0718} C_DIS
LIN {X 2.1274,Y -4.2481,Z 44,A -2.7734,B 0,C 0,E1 0.1598,E2 90.0718} C_DIS
LIN {X 2.7104,Y -3.9023,Z 44,A -2.7372,B 0,C 0,E1 0.1598,E2 90.0718} C_DIS
LIN {X 3.2392,Y -3.4779,Z 44,A -2.6997,B 0,C 0,E1 0.1598,E2 90.0718} C_DIS
LIN {X 3.699,Y -2.9797,Z 44,A -2.6616,B 0,C 0,E1 0.1598,E2 90.0718} C_DIS
LIN {X 4.0863,Y -2.4235,Z 44,A -2.6236,B 0,C 0,E1 0.1598,E2 90.0719} C_DIS
LIN {X 4.3907,Y -1.8178,Z 44,A -2.5865,B 0,C 0,E1 0.1598,E2 90.0719} C_DIS
LIN {X 4.6054,Y -1.1746,Z 44,A -2.5512,B 0,C 0,E1 0.1598,E2 90.0719} C_DIS
LIN {X 4.7225,Y -0.5069,Z 44,A -2.5184,B 0,C 0,E1 0.1598,E2 90.0719} C_DIS
LIN {X 4.7465,Y 0.1703,Z 44,A -2.4887,B 0,C 0,E1 0.1598,E2 90.0719} C_DIS
LIN {X 4.6754,Y 0.8443,Z 44,A -2.4626,B 0,C 0,E1 0.1598,E2 90.072} C_DIS
LIN {X 4.5071,Y 1.501,Z 44,A -2.4408,B 0,C 0,E1 0.1598,E2 90.072} C_DIS
LIN {X 4.2083,Y 2.2025,Z 44,A -2.4219,B 0,C 0,E1 0.1598,E2 90.072} C_DIS
LIN {X 3.901,Y 2.7098,Z 44,A -2.4117,B 0,C 0,E1 0.1598,E2 90.0722} C_DIS
LIN {X 3.4758,Y 3.2375,Z 44,A -2.4049,B 0,C 0,E1 0.1598,E2 90.0722} C_DIS
LIN {X 2.9796,Y 3.6992,Z 44,A -2.4036,B 0,C 0,E1 0.1598,E2 90.0722} C_DIS
LIN {X 2.4225,Y 4.0851,Z 44,A -2.4077,B 0,C 0,E1 0.1598,E2 90.0722} C_DIS
LIN {X 1.8171,Y 4.39,Z 44,A -2.4171,B 0,C 0,E1 0.1598,E2 90.0722} C_DIS
LIN {X 1.1742,Y 4.6048,Z 44,A -2.4317,B 0,C 0,E1 0.1598,E2 90.0722} C_DIS
LIN {X 0.507,Y 4.7258,Z 44,A -2.4512,B 0,C 0,E1 0.1598,E2 90.0722} C_DIS
LIN {X -0.1706,Y 4.7488,Z 44,A -2.4752,B 0,C 0,E1 0.1598,E2 90.0722} C_DIS
LIN {X -0.8445,Y 4.6754,Z 44,A -2.5032,B 0,C 0,E1 0.1598,E2 90.0722} C_DIS
LIN {X -1.5012,Y 4.5075,Z 44,A -2.5345,B 0,C 0,E1 0.1598,E2 90.0722} C_DIS
LIN {X -2.1274,Y 4.248,Z 44,A -2.5685,B 0,C 0,E1 0.1598,E2 90.0722} C_DIS
LIN {X -2.7098,Y 3.9013,Z 44,A -2.6047,B 0,C 0,E1 0.1598,E2 90.072} C_DIS
LIN {X -3.2375,Y 3.4759,Z 44,A -2.6421,B 0,C 0,E1 0.1598,E2 90.072} C_DIS
LIN {X -3.7003,Y 2.9806,Z 44,A -2.6801,B 0,C 0,E1 0.1598,E2 90.0719} C_DIS
LIN {X -4.086,Y 2.4232,Z 44,A -2.7179,B 0,C 0,E1 0.1598,E2 90.0718} C_DIS
LIN {X -4.3908,Y 1.8178,Z 44,A -2.7548,B 0,C 0,E1 0.1598,E2 90.0718} C_DIS
LIN {X -4.6054,Y 1.1746,Z 44,A -2.7899,B 0,C 0,E1 0.1598,E2 90.0716} C_DIS
LIN {X -4.7225,Y 0.5069,Z 44,A -2.8225,B 0,C 0,E1 0.1598,E2 90.0716} C_DIS
LIN {X -4.7465,Y -0.1703,Z 44,A -2.852,B 0,C 0,E1 0.1598,E2 90.0716} C_DIS
LIN {X -4.6746,Y -0.8442,Z 44,A -2.878,B 0,C 0,E1 0.1598,E2 90.0715} C_DIS
LIN {X -4.5082,Y -1.5013,Z 44,A -2.8997,B 0,C 0,E1 0.1598,E2 90.0715} C_DIS
LIN {X -4.2481,Y -2.1274,Z 44,A -2.9167,B 0,C 0,E1 0.1598,E2 90.0715} C_DIS
LIN {X -3.9021,Y -2.7102,Z 44,A -2.9288,B 0,C 0,E1 0.1598,E2 90.0715} C_DIS
LIN {X -3.4758,Y -3.2372,Z 44,A -2.9355,B 0,C 0,E1 0.1598,E2 90.0715} C_DIS
LIN {X -2.9796,Y -3.6989,Z 44,A -2.9369,B 0,C 0,E1 0.1598,E2 90.0715} C_DIS
LIN {X -2.4234,Y -4.0863,Z 44,A -2.933,B 0,C 0,E1 0.1598,E2 90.0715} C_DIS
LIN {X -1.8176,Y -4.3906,Z 44,A -2.9237,B 0,C 0,E1 0.1598,E2 90.0716} C_DIS
LIN {X -1.1741,Y -4.6041,Z 44,A -2.9092,B 0,C 0,E1 0.1598,E2 90.0716} C_DIS
LIN {X -0.5071,Y -4.7258,Z 44,A -2.8899,B 0,C 0,E1 0.1598,E2 90.0717} C_DIS
LIN {X -0.5071,Y -4.7258,Z 44,A -2.8899,B 0,C 0,E1 0.1598,E2 90.0717} C_DIS
Enddeposition()
LIN {X -0.0053,Y -5.6863,Z 44,A -2.9113,B 0,C 0,E1 0.1598,E2 90.0705} C_DIS
Startdeposition()
$VEL.CP = VEL_PRINT
LIN {X -0.9585,Y -5.6028,Z 44,A -2.9438,B 0,C 0,E1 0.1598,E2 90.0716} C_DIS
LIN {X -2.0216,Y -5.3185,Z 44,A -2.9708,B 0,C 0,E1 0.1598,E2 90.0716} C_DIS
LIN {X -2.5828,Y -5.064,Z 44,A -2.9806,B 0,C 0,E1 0.1598,E2 90.0716} C_DIS
LIN {X -3.2848,Y -4.6384,Z 44,A -2.9882,B 0,C 0,E1 0.1598,E2 90.0715} C_DIS
LIN {X -3.9184,Y -4.1163,Z 44,A -2.9892,B 0,C 0,E1 0.1598,E2 90.0715} C_DIS
LIN {X -4.47,Y -3.5087,Z 44,A -2.9836,B 0,C 0,E1 0.1598,E2 90.0714} C_DIS
LIN {X -4.9299,Y -2.8287,Z 44,A -2.9716,B 0,C 0,E1 0.1598,E2 90.0714} C_DIS
LIN {X -5.2844,Y -2.0883,Z 44,A -2.9532,B 0,C 0,E1 0.1598,E2 90.0714} C_DIS
LIN {X -5.5323,Y -1.3057,Z 44,A -2.9291,B 0,C 0,E1 0.1598,E2 90.0714} C_DIS
LIN {X -5.6639,Y -0.4952,Z 44,A -2.8996,B 0,C 0,E1 0.1598,E2 90.0714} C_DIS
LIN {X -5.6764,Y 0.3259,Z 44,A -2.8652,B 0,C 0,E1 0.1598,E2 90.0714} C_DIS
LIN {X -5.5688,Y 1.1399,Z 44,A -2.8268,B 0,C 0,E1 0.1598,E2 90.0714} C_DIS
LIN {X -5.3458,Y 1.9299,Z 44,A -2.7852,B 0,C 0,E1 0.1598,E2 90.0715} C_DIS
LIN {X -5.0132,Y 2.6806,Z 44,A -2.7412,B 0,C 0,E1 0.1598,E2 90.0716} C_DIS
Enddeposition()
END
